LIN {X 0,Y 171.672,Z 289.498,A -85,B 0,C 180,E1 -23440.312,E2 -23440.312} C_VEL
LIN {X 0,Y 173.108,Z 291.829,A -85,B 0,C 180,E1 -23441.183,E2 -23441.183} C_VEL
LIN {X 0,Y 175.242,Z 296.051,A -85,B 0,C 180,E1 -23442.591,E2 -23442.591} C_VEL
LIN {X 0,Y 178.721,Z 304.171,A -85,B 0,C 180,E1 -23445.058,E2 -23445.058} C_VEL
LIN {X 0,Y 180.563,Z 309.956,A -85,B 0,C 180,E1 -23446.66,E2 -23446.66} C_VEL
LIN {X 0,Y 181.625,Z 319.41,A -85,B 0,C 180,E1 -23448.871,E2 -23448.871} C_VEL
LIN {X 0,Y 181.951,Z 330.232,A -85,B 0,C 180,E1 -23451.521,E2 -23451.521} C_VEL
LIN {X 0,Y 181.208,Z 341.103,A -85,B 0,C 180,E1 -23454.43,E2 -23454.43} C_VEL
LIN {X 0,Y 179.983,Z 349.237,A -85,B 0,C 180,E1 -23456.865,E2 -23456.865} C_VEL
LIN {X 0,Y 178.407,Z 354.481,A -85,B 0,C 180,E1 -23458.54,E2 -23458.54} C_VEL
LIN {X 0,Y 174.215,Z 363.38,A -85,B 0,C 180,E1 -23461.709,E2 -23461.709} C_VEL
LIN {X 0,Y 170.995,Z 369.924,A -85,B 0,C 180,E1 -23464.717,E2 -23464.717} C_VEL
LIN {X 0,Y 168.225,Z 375.423,A -85,B 0,C 180,E1 -23467.918,E2 -23467.918} C_VEL
LIN {X 0,Y 165.735,Z 380.164,A -85,B 0,C 180,E1 -23471.46,E2 -23471.46} C_VEL
LIN {X 0,Y 163.854,Z 383.806,A -85,B 0,C 180,E1 -23475.091,E2 -23475.091} C_VEL
LIN {X 0,Y 163.072,Z 385.703,A -85,B 0,C 180,E1 -23477.56,E2 -23477.56} C_VEL
LIN {X 0,Y 162.169,Z 388.175,A -85,B 0,C 180,E1 -23482.533,E2 -23482.533} C_VEL
LIN {X 0,Y 162.078,Z 388.951,A -85,B 0,C 180,E1 -23485.808,E2 -23485.808} C_VEL
LIN {X 0,Y 162.342,Z 388.901,A -85,B 0,C 180,E1 -23490.004,E2 -23490.004} C_VEL
LIN {X 0,Y 162.14,Z 387.508,A -85,B 0,C 180,E1 -23494.483,E2 -23494.483} C_VEL
LIN {X 0,Y 162.204,Z 385.856,A -85,B 0,C 180,E1 -23497.472,E2 -23497.472} C_VEL
LIN {X 0,Y 162.769,Z 382.872,A -85,B 0,C 180,E1 -23501.207,E2 -23501.207} C_VEL
LIN {X 0,Y 163.813,Z 378.83,A -85,B 0,C 180,E1 -23504.92,E2 -23504.92} C_VEL
LIN {X 0,Y 166.011,Z 372.637,A -85,B 0,C 180,E1 -23509.157,E2 -23509.157} C_VEL
LIN {X 0,Y 168.468,Z 365.702,A -85,B 0,C 180,E1 -23512.788,E2 -23512.788} C_VEL
LIN {X 0,Y 170.299,Z 360.479,A -85,B 0,C 180,E1 -23515.028,E2 -23515.028} C_VEL
LIN {X 0,Y 171.171,Z 358.102,A -85,B 0,C 180,E1 -23515.922,E2 -23515.922} C_VEL
LIN {X 0,Y 171.863,Z 354.222,A -85,B 0,C 180,E1 -23517.39,E2 -23517.39} C_VEL
LIN {X 0,Y 171.49,Z 350.309,A -85,B 0,C 180,E1 -23518.883,E2 -23518.883} C_VEL
LIN {X 0,Y 169.685,Z 342.18,A -85,B 0,C 180,E1 -23521.821,E2 -23521.821} C_VEL
LIN {X 0,Y 169.296,Z 337.746,A -85,B 0,C 180,E1 -23523.199,E2 -23523.199} C_VEL
LIN {X 0,Y 169.37,Z 336.183,A -85,B 0,C 180,E1 -23523.629,E2 -23523.629} C_VEL
LIN {X 0,Y 169.918,Z 325.947,A -85,B 0,C 180,E1 -23526.159,E2 -23526.159} C_VEL
LIN {X 0,Y 169.626,Z 314.591,A -85,B 0,C 180,E1 -23528.627,E2 -23528.627} C_VEL
LIN {X 0,Y 168.295,Z 303.304,A -85,B 0,C 180,E1 -23530.881,E2 -23530.881} C_VEL
LIN {X 0,Y 166.877,Z 296.979,A -85,B 0,C 180,E1 -23532.153,E2 -23532.153} C_VEL
LIN {X 0,Y 163.62,Z 289.327,A -85,B 0,C 180,E1 -23534.018,E2 -23534.018} C_VEL
LIN {X 0,Y 161.492,Z 284.949,A -85,B 0,C 180,E1 -23535.128,E2 -23535.128} C_VEL
LIN {X 0,Y 159.84,Z 281.976,A -85,B 0,C 180,E1 -23535.952,E2 -23535.952} C_VEL
LIN {X 0,Y 159.355,Z 280.151,A -85,B 0,C 180,E1 -23536.332,E2 -23536.332} C_VEL
LIN {X 0,Y 158.671,Z 276.748,A -85,B 0,C 180,E1 -23541.677,E2 -23541.677} C_VEL
LIN {X 0,Y 158.331,Z 274.968,A -85,B 0,C 180,E1 -23544.757,E2 -23544.757} C_VEL
LIN {X 0,Y 157.783,Z 271.808,A -85,B 0,C 180,E1 -23550.662,E2 -23550.662} C_VEL
LIN {X 0,Y 157.407,Z 269.136,A -85,B 0,C 180,E1 -23556.307,E2 -23556.307} C_VEL
LIN {X 0,Y 157.365,Z 268.884,A -85,B 0,C 180,E1 -23559.067,E2 -23559.067} C_VEL
LIN {X 0,Y 157.424,Z 268.877,A -85,B 0,C 180,E1 -23564.463,E2 -23564.463} C_VEL
LIN {X 0,Y 157.696,Z 268.844,A -85,B 0,C 180,E1 -23569.731,E2 -23569.731} C_VEL
LIN {X 0,Y 157.773,Z 268.829,A -85,B 0,C 180,E1 -23572.321,E2 -23572.321} C_VEL
LIN {X 0,Y 158.256,Z 268.766,A -85,B 0,C 180,E1 -23580,E2 -23580} C_VEL
LIN {X 0,Y 157.768,Z 268.832,A -85,B 0,C 180,E1 -23587.68,E2 -23587.68} C_VEL
LIN {X 0,Y 157.642,Z 268.846,A -85,B 0,C 180,E1 -23591.227,E2 -23591.227} C_VEL
LIN {X 0,Y 157.428,Z 268.869,A -85,B 0,C 180,E1 -23595.537,E2 -23595.537} C_VEL
LIN {X 0,Y 157.313,Z 268.885,A -85,B 0,C 180,E1 -23600.941,E2 -23600.941} C_VEL
LIN {X 0,Y 157.275,Z 268.895,A -85,B 0,C 180,E1 -23606.648,E2 -23606.648} C_VEL
LIN {X 0,Y 157.276,Z 268.891,A -85,B 0,C 180,E1 -23612.428,E2 -23612.428} C_VEL
LIN {X 0,Y 157.276,Z 268.891,A -85,B 0,C 180,E1 -23616.447,E2 -23616.447} C_VEL
LIN {X 0,Y 157.2,Z 268.903,A -85,B 0,C 180,E1 -23622.115,E2 -23622.115} C_VEL
LIN {X 0,Y 157.242,Z 269.093,A -85,B 0,C 180,E1 -23627.561,E2 -23627.561} C_VEL
LIN {X 0,Y 158.301,Z 271.841,A -85,B 0,C 180,E1 -23628.219,E2 -23628.219} C_VEL
LIN {X 0,Y 160.043,Z 273.99,A -85,B 0,C 180,E1 -23629.056,E2 -23629.056} C_VEL
LIN {X 0,Y 162.024,Z 277.365,A -85,B 0,C 180,E1 -23630.123,E2 -23630.123} C_VEL
LIN {X 0,Y 166.172,Z 285.02,A -85,B 0,C 180,E1 -23632.468,E2 -23632.468} C_VEL
LIN {X 0,Y 169.015,Z 291.893,A -85,B 0,C 180,E1 -23634.394,E2 -23634.394} C_VEL
LIN {X 0,Y 171.62,Z 301.379,A -85,B 0,C 180,E1 -23636.891,E2 -23636.891} C_VEL
LIN {X 0,Y 173.11,Z 310.138,A -85,B 0,C 180,E1 -23639.237,E2 -23639.237} C_VEL
LIN {X 0,Y 173.769,Z 318.596,A -85,B 0,C 180,E1 -23641.622,E2 -23641.622} C_VEL
LIN {X 0,Y 171.201,Z 327.313,A -85,B 0,C 180,E1 -23643.809,E2 -23643.809} C_VEL
LIN {X 0,Y 167.929,Z 336.319,A -85,B 0,C 180,E1 -23646.569,E2 -23646.569} C_VEL
LIN {X 0,Y 164.545,Z 345.089,A -85,B 0,C 180,E1 -23650.016,E2 -23650.016} C_VEL
LIN {X 0,Y 161.778,Z 352.126,A -85,B 0,C 180,E1 -23653.594,E2 -23653.594} C_VEL
LIN {X 0,Y 159.361,Z 357.749,A -85,B 0,C 180,E1 -23657.258,E2 -23657.258} C_VEL
LIN {X 0,Y 157.576,Z 362.176,A -85,B 0,C 180,E1 -23661.016,E2 -23661.016} C_VEL
LIN {X 0,Y 156.24,Z 365.551,A -85,B 0,C 180,E1 -23664.835,E2 -23664.835} C_VEL
LIN {X 0,Y 155.458,Z 368.499,A -85,B 0,C 180,E1 -23669.996,E2 -23669.996} C_VEL
LIN {X 0,Y 155.372,Z 369.393,A -85,B 0,C 180,E1 -23672.589,E2 -23672.589} C_VEL
LIN {X 0,Y 155.479,Z 369.94,A -85,B 0,C 180,E1 -23676.032,E2 -23676.032} C_VEL
LIN {X 0,Y 155.945,Z 369.683,A -85,B 0,C 180,E1 -23680.381,E2 -23680.381} C_VEL
LIN {X 0,Y 156.512,Z 369.016,A -85,B 0,C 180,E1 -23682.971,E2 -23682.971} C_VEL
LIN {X 0,Y 157.336,Z 367.935,A -85,B 0,C 180,E1 -23685.542,E2 -23685.542} C_VEL
LIN {X 0,Y 158.403,Z 366.418,A -85,B 0,C 180,E1 -23688.09,E2 -23688.09} C_VEL
LIN {X 0,Y 160.603,Z 363.348,A -85,B 0,C 180,E1 -23691.833,E2 -23691.833} C_VEL
LIN {X 0,Y 163.269,Z 359.22,A -85,B 0,C 180,E1 -23695.492,E2 -23695.492} C_VEL
LIN {X 0,Y 167.172,Z 352.9,A -85,B 0,C 180,E1 -23699.598,E2 -23699.598} C_VEL
LIN {X 0,Y 171.048,Z 345.979,A -85,B 0,C 180,E1 -23702.98,E2 -23702.98} C_VEL
LIN {X 0,Y 175.423,Z 337.268,A -85,B 0,C 180,E1 -23706.219,E2 -23706.219} C_VEL
LIN {X 0,Y 179.363,Z 328.323,A -85,B 0,C 180,E1 -23708.82,E2 -23708.82} C_VEL
LIN {X 0,Y 179.655,Z 326.596,A -85,B 0,C 180,E1 -23709.372,E2 -23709.372} C_VEL
LIN {X 0,Y 179.152,Z 317.685,A -85,B 0,C 180,E1 -23712.437,E2 -23712.437} C_VEL
LIN {X 0,Y 177.698,Z 308.9,A -85,B 0,C 180,E1 -23715.385,E2 -23715.385} C_VEL
LIN {X 0,Y 175.607,Z 301.826,A -85,B 0,C 180,E1 -23717.854,E2 -23717.854} C_VEL
LIN {X 0,Y 171.735,Z 292.618,A -85,B 0,C 180,E1 -23721.343,E2 -23721.343} C_VEL
LIN {X 0,Y 167.163,Z 284.059,A -85,B 0,C 180,E1 -23724.96,E2 -23724.96} C_VEL
LIN {X 0,Y 164.783,Z 280.149,A -85,B 0,C 180,E1 -23726.784,E2 -23726.784} C_VEL
LIN {X 0,Y 161.938,Z 276.182,A -85,B 0,C 180,E1 -23728.895,E2 -23728.895} C_VEL
LIN {X 0,Y 161.277,Z 274.774,A -85,B 0,C 180,E1 -23729.48,E2 -23729.48} C_VEL
LIN {X 0,Y 158.718,Z 272.463,A -85,B 0,C 180,E1 -23731.304,E2 -23731.304} C_VEL
LIN {X 0,Y 157.479,Z 269.821,A -85,B 0,C 180,E1 -23732.455,E2 -23732.455} C_VEL
LIN {X 0,Y 157.37,Z 269.368,A -85,B 0,C 180,E1 -23732.632,E2 -23732.632} C_VEL
LIN {X 0,Y 157.304,Z 268.891,A -85,B 0,C 180,E1 -23736.29,E2 -23736.29} C_VEL
LIN {X 0,Y 157.402,Z 268.876,A -85,B 0,C 180,E1 -23741.787,E2 -23741.787} C_VEL
LIN {X 0,Y 157.544,Z 268.861,A -85,B 0,C 180,E1 -23747.111,E2 -23747.111} C_VEL
LIN {X 0,Y 157.763,Z 268.835,A -85,B 0,C 180,E1 -23749.735,E2 -23749.735} C_VEL
LIN {X 0,Y 157.815,Z 268.828,A -85,B 0,C 180,E1 -23752.322,E2 -23752.322} C_VEL
LIN {X 0,Y 158.004,Z 268.803,A -85,B 0,C 180,E1 -23757.45,E2 -23757.45} C_VEL
LIN {X 0,Y 158.246,Z 268.772,A -85,B 0,C 180,E1 -23760,E2 -23760} C_VEL
LIN {X 0,Y 157.723,Z 268.862,A -85,B 0,C 180,E1 -23765.113,E2 -23765.113} C_VEL
LIN {X 0,Y 157.962,Z 269.906,A -85,B 0,C 180,E1 -23770.251,E2 -23770.251} C_VEL
LIN {X 0,Y 157.918,Z 271.393,A -85,B 0,C 180,E1 -23775.487,E2 -23775.487} C_VEL
LIN {X 0,Y 158.171,Z 273.297,A -85,B 0,C 180,E1 -23781.09,E2 -23781.09} C_VEL
LIN {X 0,Y 158.588,Z 275.985,A -85,B 0,C 180,E1 -23787.595,E2 -23787.595} C_VEL
LIN {X 0,Y 158.956,Z 278.479,A -85,B 0,C 180,E1 -23792.725,E2 -23792.725} C_VEL
LIN {X 0,Y 160.11,Z 281.618,A -85,B 0,C 180,E1 -23793.767,E2 -23793.767} C_VEL
LIN {X 0,Y 162.377,Z 284.59,A -85,B 0,C 180,E1 -23795.373,E2 -23795.373} C_VEL
LIN {X 0,Y 163.054,Z 285.722,A -85,B 0,C 180,E1 -23795.862,E2 -23795.862} C_VEL
LIN {X 0,Y 164.865,Z 289.444,A -85,B 0,C 180,E1 -23797.29,E2 -23797.29} C_VEL
LIN {X 0,Y 166.299,Z 291.666,A -85,B 0,C 180,E1 -23798.272,E2 -23798.272} C_VEL
LIN {X 0,Y 168.363,Z 295.763,A -85,B 0,C 180,E1 -23799.829,E2 -23799.829} C_VEL
LIN {X 0,Y 171.594,Z 302.812,A -85,B 0,C 180,E1 -23802.316,E2 -23802.316} C_VEL
LIN {X 0,Y 174.732,Z 311.358,A -85,B 0,C 180,E1 -23805.082,E2 -23805.082} C_VEL
LIN {X 0,Y 175.6,Z 316.698,A -85,B 0,C 180,E1 -23806.503,E2 -23806.503} C_VEL
LIN {X 0,Y 176.02,Z 327.827,A -85,B 0,C 180,E1 -23809.342,E2 -23809.342} C_VEL
LIN {X 0,Y 175.468,Z 337.565,A -85,B 0,C 180,E1 -23811.994,E2 -23811.994} C_VEL
LIN {X 0,Y 174.366,Z 346.244,A -85,B 0,C 180,E1 -23814.625,E2 -23814.625} C_VEL
LIN {X 0,Y 172.964,Z 352.639,A -85,B 0,C 180,E1 -23816.737,E2 -23816.737} C_VEL
LIN {X 0,Y 170.1,Z 358.951,A -85,B 0,C 180,E1 -23818.909,E2 -23818.909} C_VEL
LIN {X 0,Y 166.033,Z 366.907,A -85,B 0,C 180,E1 -23822.254,E2 -23822.254} C_VEL
LIN {X 0,Y 162.685,Z 373.292,A -85,B 0,C 180,E1 -23825.774,E2 -23825.774} C_VEL
LIN {X 0,Y 159.795,Z 378.389,A -85,B 0,C 180,E1 -23829.404,E2 -23829.404} C_VEL
LIN {X 0,Y 157.566,Z 382.364,A -85,B 0,C 180,E1 -23833.151,E2 -23833.151} C_VEL
LIN {X 0,Y 156.091,Z 385.326,A -85,B 0,C 180,E1 -23836.994,E2 -23836.994} C_VEL
LIN {X 0,Y 155.109,Z 387.774,A -85,B 0,C 180,E1 -23842.191,E2 -23842.191} C_VEL
LIN {X 0,Y 155.007,Z 388.553,A -85,B 0,C 180,E1 -23845.927,E2 -23845.927} C_VEL
LIN {X 0,Y 155.254,Z 388.457,A -85,B 0,C 180,E1 -23850.004,E2 -23850.004} C_VEL
LIN {X 0,Y 155.075,Z 387.163,A -85,B 0,C 180,E1 -23854.412,E2 -23854.412} C_VEL
LIN {X 0,Y 155.159,Z 385.37,A -85,B 0,C 180,E1 -23857.814,E2 -23857.814} C_VEL
LIN {X 0,Y 155.79,Z 382.365,A -85,B 0,C 180,E1 -23861.716,E2 -23861.716} C_VEL
LIN {X 0,Y 156.919,Z 378.296,A -85,B 0,C 180,E1 -23865.592,E2 -23865.592} C_VEL
LIN {X 0,Y 159.261,Z 372.063,A -85,B 0,C 180,E1 -23870.002,E2 -23870.002} C_VEL
LIN {X 0,Y 161.71,Z 365.444,A -85,B 0,C 180,E1 -23873.606,E2 -23873.606} C_VEL
LIN {X 0,Y 164.999,Z 356.823,A -85,B 0,C 180,E1 -23877.255,E2 -23877.255} C_VEL
LIN {X 0,Y 167.455,Z 349.995,A -85,B 0,C 180,E1 -23879.551,E2 -23879.551} C_VEL
LIN {X 0,Y 168.915,Z 340.714,A -85,B 0,C 180,E1 -23882.394,E2 -23882.394} C_VEL
LIN {X 0,Y 169.37,Z 336.183,A -85,B 0,C 180,E1 -23883.629,E2 -23883.629} C_VEL
LIN {X 0,Y 169.123,Z 331.677,A -85,B 0,C 180,E1 -23884.918,E2 -23884.918} C_VEL
LIN {X 0,Y 166.874,Z 324.632,A -85,B 0,C 180,E1 -23887.172,E2 -23887.172} C_VEL
LIN {X 0,Y 164.677,Z 318.905,A -85,B 0,C 180,E1 -23888.963,E2 -23888.963} C_VEL
LIN {X 0,Y 163.523,Z 314.238,A -85,B 0,C 180,E1 -23890.21,E2 -23890.21} C_VEL
LIN {X 0,Y 163.305,Z 312.574,A -85,B 0,C 180,E1 -23890.589,E2 -23890.589} C_VEL
LIN {X 0,Y 162.2,Z 303.334,A -85,B 0,C 180,E1 -23892.558,E2 -23892.558} C_VEL
LIN {X 0,Y 160.439,Z 297.745,A -85,B 0,C 180,E1 -23893.942,E2 -23893.942} C_VEL
LIN {X 0,Y 156.925,Z 289.667,A -85,B 0,C 180,E1 -23896.148,E2 -23896.148} C_VEL
LIN {X 0,Y 155.023,Z 285.715,A -85,B 0,C 180,E1 -23897.275,E2 -23897.275} C_VEL
LIN {X 0,Y 152.557,Z 281.546,A -85,B 0,C 180,E1 -23898.625,E2 -23898.625} C_VEL
LIN {X 0,Y 151.956,Z 279.532,A -85,B 0,C 180,E1 -23899.094,E2 -23899.094} C_VEL
LIN {X 0,Y 151.576,Z 277.292,A -85,B 0,C 180,E1 -23902.932,E2 -23902.932} C_VEL
LIN {X 0,Y 150.916,Z 273.997,A -85,B 0,C 180,E1 -23909.186,E2 -23909.186} C_VEL
LIN {X 0,Y 150.529,Z 271.205,A -85,B 0,C 180,E1 -23915.153,E2 -23915.153} C_VEL
LIN {X 0,Y 150.327,Z 269.76,A -85,B 0,C 180,E1 -23918.801,E2 -23918.801} C_VEL
LIN {X 0,Y 150.333,Z 269.762,A -85,B 0,C 180,E1 -23923.71,E2 -23923.71} C_VEL
LIN {X 0,Y 150.616,Z 269.726,A -85,B 0,C 180,E1 -23929.243,E2 -23929.243} C_VEL
LIN {X 0,Y 150.711,Z 269.709,A -85,B 0,C 180,E1 -23931.958,E2 -23931.958} C_VEL
LIN {X 0,Y 151.215,Z 269.643,A -85,B 0,C 180,E1 -23940,E2 -23940} C_VEL
LIN {X 0,Y 150.691,Z 269.713,A -85,B 0,C 180,E1 -23948.043,E2 -23948.043} C_VEL
LIN {X 0,Y 150.584,Z 269.726,A -85,B 0,C 180,E1 -23951.43,E2 -23951.43} C_VEL
LIN {X 0,Y 150.333,Z 269.757,A -85,B 0,C 180,E1 -23956.29,E2 -23956.29} C_VEL
LIN {X 0,Y 150.291,Z 269.758,A -85,B 0,C 180,E1 -23960.721,E2 -23960.721} C_VEL
LIN {X 0,Y 150.193,Z 269.776,A -85,B 0,C 180,E1 -23967.236,E2 -23967.236} C_VEL
LIN {X 0,Y 150.217,Z 269.769,A -85,B 0,C 180,E1 -23972.626,E2 -23972.626} C_VEL
LIN {X 0,Y 150.186,Z 269.774,A -85,B 0,C 180,E1 -23977.47,E2 -23977.47} C_VEL
LIN {X 0,Y 150.145,Z 269.783,A -85,B 0,C 180,E1 -23981.497,E2 -23981.497} C_VEL
LIN {X 0,Y 150.132,Z 269.793,A -85,B 0,C 180,E1 -23984.818,E2 -23984.818} C_VEL
LIN {X 0,Y 151.135,Z 272.602,A -85,B 0,C 180,E1 -23985.545,E2 -23985.545} C_VEL
LIN {X 0,Y 153.242,Z 275.172,A -85,B 0,C 180,E1 -23986.696,E2 -23986.696} C_VEL
LIN {X 0,Y 155.261,Z 278.518,A -85,B 0,C 180,E1 -23987.896,E2 -23987.896} C_VEL
LIN {X 0,Y 159.442,Z 285.905,A -85,B 0,C 180,E1 -23990.479,E2 -23990.479} C_VEL
LIN {X 0,Y 163.192,Z 294.405,A -85,B 0,C 180,E1 -23993.16,E2 -23993.16} C_VEL
LIN {X 0,Y 165.754,Z 304.364,A -85,B 0,C 180,E1 -23996,E2 -23996} C_VEL
LIN {X 0,Y 167.084,Z 313.779,A -85,B 0,C 180,E1 -23998.723,E2 -23998.723} C_VEL
LIN {X 0,Y 167.338,Z 320.547,A -85,B 0,C 180,E1 -24000.771,E2 -24000.771} C_VEL
LIN {X 0,Y 164.211,Z 329.985,A -85,B 0,C 180,E1 -24003.292,E2 -24003.292} C_VEL
LIN {X 0,Y 160.844,Z 338.618,A -85,B 0,C 180,E1 -24006.157,E2 -24006.157} C_VEL
LIN {X 0,Y 157.478,Z 346.868,A -85,B 0,C 180,E1 -24009.691,E2 -24009.691} C_VEL
LIN {X 0,Y 154.527,Z 353.718,A -85,B 0,C 180,E1 -24013.482,E2 -24013.482} C_VEL
LIN {X 0,Y 151.754,Z 359.903,A -85,B 0,C 180,E1 -24017.967,E2 -24017.967} C_VEL
LIN {X 0,Y 150.022,Z 363.938,A -85,B 0,C 180,E1 -24021.917,E2 -24021.917} C_VEL
LIN {X 0,Y 149.203,Z 366.048,A -85,B 0,C 180,E1 -24024.59,E2 -24024.59} C_VEL
LIN {X 0,Y 148.393,Z 368.97,A -85,B 0,C 180,E1 -24029.996,E2 -24029.996} C_VEL
LIN {X 0,Y 148.29,Z 369.852,A -85,B 0,C 180,E1 -24032.712,E2 -24032.712} C_VEL
LIN {X 0,Y 148.377,Z 370.348,A -85,B 0,C 180,E1 -24035.907,E2 -24035.907} C_VEL
LIN {X 0,Y 148.947,Z 370.092,A -85,B 0,C 180,E1 -24040.875,E2 -24040.875} C_VEL
LIN {X 0,Y 149.581,Z 369.412,A -85,B 0,C 180,E1 -24043.583,E2 -24043.583} C_VEL
LIN {X 0,Y 150.485,Z 368.305,A -85,B 0,C 180,E1 -24046.269,E2 -24046.269} C_VEL
LIN {X 0,Y 151.634,Z 366.775,A -85,B 0,C 180,E1 -24048.927,E2 -24048.927} C_VEL
LIN {X 0,Y 153.998,Z 363.677,A -85,B 0,C 180,E1 -24052.82,E2 -24052.82} C_VEL
LIN {X 0,Y 156.846,Z 359.518,A -85,B 0,C 180,E1 -24056.616,E2 -24056.616} C_VEL
LIN {X 0,Y 160.997,Z 353.165,A -85,B 0,C 180,E1 -24060.854,E2 -24060.854} C_VEL
LIN {X 0,Y 165.104,Z 346.191,A -85,B 0,C 180,E1 -24064.329,E2 -24064.329} C_VEL
LIN {X 0,Y 169.701,Z 337.433,A -85,B 0,C 180,E1 -24067.647,E2 -24067.647} C_VEL
LIN {X 0,Y 172.997,Z 330.392,A -85,B 0,C 180,E1 -24069.771,E2 -24069.771} C_VEL
LIN {X 0,Y 173.468,Z 328.442,A -85,B 0,C 180,E1 -24070.404,E2 -24070.404} C_VEL
LIN {X 0,Y 173.178,Z 319.713,A -85,B 0,C 180,E1 -24073.617,E2 -24073.617} C_VEL
LIN {X 0,Y 172,Z 311.869,A -85,B 0,C 180,E1 -24076.459,E2 -24076.459} C_VEL
LIN {X 0,Y 170.42,Z 305.944,A -85,B 0,C 180,E1 -24078.713,E2 -24078.713} C_VEL
LIN {X 0,Y 166.952,Z 296.993,A -85,B 0,C 180,E1 -24082.382,E2 -24082.382} C_VEL
LIN {X 0,Y 163.073,Z 289.262,A -85,B 0,C 180,E1 -24085.925,E2 -24085.925} C_VEL
LIN {X 0,Y 160.476,Z 284.822,A -85,B 0,C 180,E1 -24088.203,E2 -24088.203} C_VEL
LIN {X 0,Y 158.469,Z 281.585,A -85,B 0,C 180,E1 -24089.979,E2 -24089.979} C_VEL
LIN {X 0,Y 157.694,Z 280.571,A -85,B 0,C 180,E1 -24090.643,E2 -24090.643} C_VEL
LIN {X 0,Y 155.374,Z 277.702,A -85,B 0,C 180,E1 -24092.636,E2 -24092.636} C_VEL
LIN {X 0,Y 154.407,Z 275.643,A -85,B 0,C 180,E1 -24093.678,E2 -24093.678} C_VEL
LIN {X 0,Y 151.842,Z 273.481,A -85,B 0,C 180,E1 -24095.927,E2 -24095.927} C_VEL
LIN {X 0,Y 150.46,Z 270.803,A -85,B 0,C 180,E1 -24097.515,E2 -24097.515} C_VEL
LIN {X 0,Y 150.336,Z 270.24,A -85,B 0,C 180,E1 -24097.857,E2 -24097.857} C_VEL
LIN {X 0,Y 150.351,Z 269.891,A -85,B 0,C 180,E1 -24100.9,E2 -24100.9} C_VEL
LIN {X 0,Y 150.446,Z 269.743,A -85,B 0,C 180,E1 -24106.492,E2 -24106.492} C_VEL
LIN {X 0,Y 150.679,Z 269.715,A -85,B 0,C 180,E1 -24109.247,E2 -24109.247} C_VEL
LIN {X 0,Y 150.754,Z 269.708,A -85,B 0,C 180,E1 -24111.96,E2 -24111.96} C_VEL
LIN {X 0,Y 150.927,Z 269.685,A -85,B 0,C 180,E1 -24117.331,E2 -24117.331} C_VEL
LIN {X 0,Y 151.209,Z 269.803,A -85,B 0,C 180,E1 -24120,E2 -24120} C_VEL
LIN {X 0,Y 150.991,Z 271.195,A -85,B 0,C 180,E1 -24128.027,E2 -24128.027} C_VEL
LIN {X 0,Y 151.02,Z 272.193,A -85,B 0,C 180,E1 -24132.259,E2 -24132.259} C_VEL
LIN {X 0,Y 151.147,Z 274.23,A -85,B 0,C 180,E1 -24138.995,E2 -24138.995} C_VEL
LIN {X 0,Y 151.43,Z 276.319,A -85,B 0,C 180,E1 -24144.689,E2 -24144.689} C_VEL
LIN {X 0,Y 151.662,Z 277.586,A -85,B 0,C 180,E1 -24147.693,E2 -24147.693} C_VEL
LIN {X 0,Y 152.652,Z 280.447,A -85,B 0,C 180,E1 -24148.845,E2 -24148.845} C_VEL
LIN {X 0,Y 154.921,Z 283.56,A -85,B 0,C 180,E1 -24150.877,E2 -24150.877} C_VEL
LIN {X 0,Y 155.929,Z 284.728,A -85,B 0,C 180,E1 -24151.693,E2 -24151.693} C_VEL
LIN {X 0,Y 157.57,Z 288.461,A -85,B 0,C 180,E1 -24153.303,E2 -24153.303} C_VEL
LIN {X 0,Y 159.432,Z 291.108,A -85,B 0,C 180,E1 -24154.777,E2 -24154.777} C_VEL
LIN {X 0,Y 161.439,Z 295.308,A -85,B 0,C 180,E1 -24156.574,E2 -24156.574} C_VEL
LIN {X 0,Y 162.344,Z 296.942,A -85,B 0,C 180,E1 -24157.306,E2 -24157.306} C_VEL
LIN {X 0,Y 165.552,Z 304.184,A -85,B 0,C 180,E1 -24160.176,E2 -24160.176} C_VEL
LIN {X 0,Y 168.337,Z 311.392,A -85,B 0,C 180,E1 -24162.834,E2 -24162.834} C_VEL
LIN {X 0,Y 169.856,Z 317.061,A -85,B 0,C 180,E1 -24164.7,E2 -24164.7} C_VEL
LIN {X 0,Y 170.178,Z 325.932,A -85,B 0,C 180,E1 -24167.102,E2 -24167.102} C_VEL
LIN {X 0,Y 169.814,Z 335.14,A -85,B 0,C 180,E1 -24169.726,E2 -24169.726} C_VEL
LIN {X 0,Y 168.441,Z 345.291,A -85,B 0,C 180,E1 -24172.879,E2 -24172.879} C_VEL
LIN {X 0,Y 166.88,Z 352.441,A -85,B 0,C 180,E1 -24175.356,E2 -24175.356} C_VEL
LIN {X 0,Y 164.86,Z 357.242,A -85,B 0,C 180,E1 -24177.08,E2 -24177.08} C_VEL
LIN {X 0,Y 160.41,Z 365.418,A -85,B 0,C 180,E1 -24180.474,E2 -24180.474} C_VEL
LIN {X 0,Y 157.261,Z 371.005,A -85,B 0,C 180,E1 -24183.459,E2 -24183.459} C_VEL
LIN {X 0,Y 154.054,Z 376.489,A -85,B 0,C 180,E1 -24187.188,E2 -24187.188} C_VEL
LIN {X 0,Y 151.489,Z 380.801,A -85,B 0,C 180,E1 -24191.054,E2 -24191.054} C_VEL
LIN {X 0,Y 150.09,Z 383.097,A -85,B 0,C 180,E1 -24193.687,E2 -24193.687} C_VEL
LIN {X 0,Y 149.133,Z 384.948,A -85,B 0,C 180,E1 -24196.375,E2 -24196.375} C_VEL
LIN {X 0,Y 148.042,Z 387.373,A -85,B 0,C 180,E1 -24201.816,E2 -24201.816} C_VEL
LIN {X 0,Y 147.939,Z 388.156,A -85,B 0,C 180,E1 -24206.054,E2 -24206.054} C_VEL
LIN {X 0,Y 148.168,Z 388.013,A -85,B 0,C 180,E1 -24210.004,E2 -24210.004} C_VEL
LIN {X 0,Y 147.991,Z 386.862,A -85,B 0,C 180,E1 -24214.228,E2 -24214.228} C_VEL
LIN {X 0,Y 148.093,Z 384.879,A -85,B 0,C 180,E1 -24218.189,E2 -24218.189} C_VEL
LIN {X 0,Y 148.786,Z 381.851,A -85,B 0,C 180,E1 -24222.276,E2 -24222.276} C_VEL
LIN {X 0,Y 150.054,Z 377.758,A -85,B 0,C 180,E1 -24226.325,E2 -24226.325} C_VEL
LIN {X 0,Y 152.528,Z 371.485,A -85,B 0,C 180,E1 -24230.926,E2 -24230.926} C_VEL
LIN {X 0,Y 154.789,Z 365.901,A -85,B 0,C 180,E1 -24234.123,E2 -24234.123} C_VEL
LIN {X 0,Y 156.356,Z 361.818,A -85,B 0,C 180,E1 -24236.096,E2 -24236.096} C_VEL
LIN {X 0,Y 159.954,Z 352.877,A -85,B 0,C 180,E1 -24239.628,E2 -24239.628} C_VEL
LIN {X 0,Y 161.145,Z 349.295,A -85,B 0,C 180,E1 -24240.831,E2 -24240.831} C_VEL
LIN {X 0,Y 162.618,Z 339.938,A -85,B 0,C 180,E1 -24243.813,E2 -24243.813} C_VEL
LIN {X 0,Y 163.553,Z 329.5,A -85,B 0,C 180,E1 -24246.651,E2 -24246.651} C_VEL
LIN {X 0,Y 163.643,Z 318.065,A -85,B 0,C 180,E1 -24249.372,E2 -24249.372} C_VEL
LIN {X 0,Y 163.305,Z 312.574,A -85,B 0,C 180,E1 -24250.589,E2 -24250.589} C_VEL
LIN {X 0,Y 162.672,Z 309.405,A -85,B 0,C 180,E1 -24251.375,E2 -24251.375} C_VEL
LIN {X 0,Y 160.725,Z 305.247,A -85,B 0,C 180,E1 -24252.704,E2 -24252.704} C_VEL
LIN {X 0,Y 158.118,Z 301.619,A -85,B 0,C 180,E1 -24254.135,E2 -24254.135} C_VEL
LIN {X 0,Y 152.492,Z 294.366,A -85,B 0,C 180,E1 -24257.13,E2 -24257.13} C_VEL
LIN {X 0,Y 150.966,Z 291.539,A -85,B 0,C 180,E1 -24258.072,E2 -24258.072} C_VEL
LIN {X 0,Y 149.674,Z 289.051,A -85,B 0,C 180,E1 -24258.9,E2 -24258.9} C_VEL
LIN {X 0,Y 147.872,Z 285.19,A -85,B 0,C 180,E1 -24260.127,E2 -24260.127} C_VEL
LIN {X 0,Y 145.314,Z 281.196,A -85,B 0,C 180,E1 -24261.694,E2 -24261.694} C_VEL
LIN {X 0,Y 144.668,Z 278.923,A -85,B 0,C 180,E1 -24262.28,E2 -24262.28} C_VEL
LIN {X 0,Y 144.086,Z 276.201,A -85,B 0,C 180,E1 -24267.552,E2 -24267.552} C_VEL
LIN {X 0,Y 143.648,Z 273.294,A -85,B 0,C 180,E1 -24273.876,E2 -24273.876} C_VEL
LIN {X 0,Y 143.33,Z 270.88,A -85,B 0,C 180,E1 -24279.926,E2 -24279.926} C_VEL
LIN {X 0,Y 143.273,Z 270.639,A -85,B 0,C 180,E1 -24282.884,E2 -24282.884} C_VEL
LIN {X 0,Y 143.542,Z 270.608,A -85,B 0,C 180,E1 -24288.706,E2 -24288.706} C_VEL
LIN {X 0,Y 143.632,Z 270.592,A -85,B 0,C 180,E1 -24291.559,E2 -24291.559} C_VEL
LIN {X 0,Y 144.172,Z 270.52,A -85,B 0,C 180,E1 -24300,E2 -24300} C_VEL
LIN {X 0,Y 143.616,Z 270.592,A -85,B 0,C 180,E1 -24308.442,E2 -24308.442} C_VEL
LIN {X 0,Y 143.51,Z 270.608,A -85,B 0,C 180,E1 -24311.618,E2 -24311.618} C_VEL
LIN {X 0,Y 143.27,Z 270.64,A -85,B 0,C 180,E1 -24317.118,E2 -24317.118} C_VEL
LIN {X 0,Y 143.228,Z 270.641,A -85,B 0,C 180,E1 -24321.193,E2 -24321.193} C_VEL
LIN {X 0,Y 143.151,Z 270.651,A -85,B 0,C 180,E1 -24327.898,E2 -24327.898} C_VEL
LIN {X 0,Y 143.148,Z 270.649,A -85,B 0,C 180,E1 -24333.415,E2 -24333.415} C_VEL
LIN {X 0,Y 143.065,Z 270.661,A -85,B 0,C 180,E1 -24339.69,E2 -24339.69} C_VEL
LIN {X 0,Y 143.114,Z 270.73,A -85,B 0,C 180,E1 -24341.697,E2 -24341.697} C_VEL
LIN {X 0,Y 143.928,Z 273.29,A -85,B 0,C 180,E1 -24342.409,E2 -24342.409} C_VEL
LIN {X 0,Y 145.881,Z 275.494,A -85,B 0,C 180,E1 -24343.616,E2 -24343.616} C_VEL
LIN {X 0,Y 148.362,Z 279.492,A -85,B 0,C 180,E1 -24345.281,E2 -24345.281} C_VEL
LIN {X 0,Y 149.478,Z 281.345,A -85,B 0,C 180,E1 -24346.048,E2 -24346.048} C_VEL
LIN {X 0,Y 152.84,Z 287.147,A -85,B 0,C 180,E1 -24348.351,E2 -24348.351} C_VEL
LIN {X 0,Y 156.345,Z 294.484,A -85,B 0,C 180,E1 -24350.995,E2 -24350.995} C_VEL
LIN {X 0,Y 158.088,Z 299.409,A -85,B 0,C 180,E1 -24352.623,E2 -24352.623} C_VEL
LIN {X 0,Y 160.107,Z 308.638,A -85,B 0,C 180,E1 -24355.486,E2 -24355.486} C_VEL
LIN {X 0,Y 160.998,Z 317.978,A -85,B 0,C 180,E1 -24358.406,E2 -24358.406} C_VEL
LIN {X 0,Y 161.099,Z 321.365,A -85,B 0,C 180,E1 -24359.522,E2 -24359.522} C_VEL
LIN {X 0,Y 158.654,Z 328.792,A -85,B 0,C 180,E1 -24361.559,E2 -24361.559} C_VEL
LIN {X 0,Y 155.08,Z 337.693,A -85,B 0,C 180,E1 -24364.495,E2 -24364.495} C_VEL
LIN {X 0,Y 151.207,Z 346.744,A -85,B 0,C 180,E1 -24368.372,E2 -24368.372} C_VEL
LIN {X 0,Y 147.781,Z 354.305,A -85,B 0,C 180,E1 -24372.705,E2 -24372.705} C_VEL
LIN {X 0,Y 144.854,Z 360.458,A -85,B 0,C 180,E1 -24377.385,E2 -24377.385} C_VEL
LIN {X 0,Y 143.031,Z 364.463,A -85,B 0,C 180,E1 -24381.519,E2 -24381.519} C_VEL
LIN {X 0,Y 142.17,Z 366.546,A -85,B 0,C 180,E1 -24384.322,E2 -24384.322} C_VEL
LIN {X 0,Y 141.328,Z 369.441,A -85,B 0,C 180,E1 -24389.996,E2 -24389.996} C_VEL
LIN {X 0,Y 141.211,Z 370.308,A -85,B 0,C 180,E1 -24392.849,E2 -24392.849} C_VEL
LIN {X 0,Y 141.297,Z 370.76,A -85,B 0,C 180,E1 -24395.85,E2 -24395.85} C_VEL
LIN {X 0,Y 141.955,Z 370.502,A -85,B 0,C 180,E1 -24401.418,E2 -24401.418} C_VEL
LIN {X 0,Y 142.663,Z 369.807,A -85,B 0,C 180,E1 -24404.255,E2 -24404.255} C_VEL
LIN {X 0,Y 143.645,Z 368.675,A -85,B 0,C 180,E1 -24407.067,E2 -24407.067} C_VEL
LIN {X 0,Y 144.899,Z 367.132,A -85,B 0,C 180,E1 -24409.843,E2 -24409.843} C_VEL
LIN {X 0,Y 147.445,Z 364.006,A -85,B 0,C 180,E1 -24413.896,E2 -24413.896} C_VEL
LIN {X 0,Y 150.493,Z 359.817,A -85,B 0,C 180,E1 -24417.835,E2 -24417.835} C_VEL
LIN {X 0,Y 154.915,Z 353.432,A -85,B 0,C 180,E1 -24422.208,E2 -24422.208} C_VEL
LIN {X 0,Y 159.274,Z 346.401,A -85,B 0,C 180,E1 -24425.774,E2 -24425.774} C_VEL
LIN {X 0,Y 164.09,Z 337.6,A -85,B 0,C 180,E1 -24429.174,E2 -24429.174} C_VEL
LIN {X 0,Y 166.671,Z 332.4,A -85,B 0,C 180,E1 -24430.813,E2 -24430.813} C_VEL
LIN {X 0,Y 167.32,Z 330.496,A -85,B 0,C 180,E1 -24431.416,E2 -24431.416} C_VEL
LIN {X 0,Y 167.321,Z 322.867,A -85,B 0,C 180,E1 -24434.434,E2 -24434.434} C_VEL
LIN {X 0,Y 166.4,Z 315.113,A -85,B 0,C 180,E1 -24437.485,E2 -24437.485} C_VEL
LIN {X 0,Y 164.725,Z 308.535,A -85,B 0,C 180,E1 -24440.209,E2 -24440.209} C_VEL
LIN {X 0,Y 161.839,Z 300.594,A -85,B 0,C 180,E1 -24443.783,E2 -24443.783} C_VEL
LIN {X 0,Y 159.146,Z 294.821,A -85,B 0,C 180,E1 -24446.646,E2 -24446.646} C_VEL
LIN {X 0,Y 156.857,Z 290.574,A -85,B 0,C 180,E1 -24448.985,E2 -24448.985} C_VEL
LIN {X 0,Y 154.258,Z 286.367,A -85,B 0,C 180,E1 -24451.605,E2 -24451.605} C_VEL
LIN {X 0,Y 152.128,Z 283.217,A -85,B 0,C 180,E1 -24453.783,E2 -24453.783} C_VEL
LIN {X 0,Y 151.474,Z 281.878,A -85,B 0,C 180,E1 -24454.584,E2 -24454.584} C_VEL
LIN {X 0,Y 149.227,Z 279.589,A -85,B 0,C 180,E1 -24456.861,E2 -24456.861} C_VEL
LIN {X 0,Y 147.772,Z 276.734,A -85,B 0,C 180,E1 -24458.8,E2 -24458.8} C_VEL
LIN {X 0,Y 144.693,Z 274.141,A -85,B 0,C 180,E1 -24462.51,E2 -24462.51} C_VEL
LIN {X 0,Y 143.505,Z 271.609,A -85,B 0,C 180,E1 -24464.556,E2 -24464.556} C_VEL
LIN {X 0,Y 143.457,Z 271.335,A -85,B 0,C 180,E1 -24465.096,E2 -24465.096} C_VEL
LIN {X 0,Y 143.7,Z 271.158,A -85,B 0,C 180,E1 -24468.718,E2 -24468.718} C_VEL
LIN {X 0,Y 143.769,Z 271.156,A -85,B 0,C 180,E1 -24471.567,E2 -24471.567} C_VEL
LIN {X 0,Y 144.025,Z 271.397,A -85,B 0,C 180,E1 -24477.203,E2 -24477.203} C_VEL
LIN {X 0,Y 144.331,Z 271.606,A -85,B 0,C 180,E1 -24480,E2 -24480} C_VEL
LIN {X 0,Y 144.098,Z 273.036,A -85,B 0,C 180,E1 -24488.413,E2 -24488.413} C_VEL
LIN {X 0,Y 144.113,Z 274.074,A -85,B 0,C 180,E1 -24492.77,E2 -24492.77} C_VEL
LIN {X 0,Y 144.13,Z 275.273,A -85,B 0,C 180,E1 -24497.012,E2 -24497.012} C_VEL
LIN {X 0,Y 144.323,Z 276.57,A -85,B 0,C 180,E1 -24500.72,E2 -24500.72} C_VEL
LIN {X 0,Y 145.754,Z 280.144,A -85,B 0,C 180,E1 -24502.971,E2 -24502.971} C_VEL
LIN {X 0,Y 148.748,Z 283.606,A -85,B 0,C 180,E1 -24506.348,E2 -24506.348} C_VEL
LIN {X 0,Y 150.902,Z 288.221,A -85,B 0,C 180,E1 -24508.945,E2 -24508.945} C_VEL
LIN {X 0,Y 152.739,Z 290.649,A -85,B 0,C 180,E1 -24510.694,E2 -24510.694} C_VEL
LIN {X 0,Y 154.454,Z 294.581,A -85,B 0,C 180,E1 -24512.61,E2 -24512.61} C_VEL
LIN {X 0,Y 155.587,Z 296.14,A -85,B 0,C 180,E1 -24513.596,E2 -24513.596} C_VEL
LIN {X 0,Y 157.339,Z 300.365,A -85,B 0,C 180,E1 -24515.498,E2 -24515.498} C_VEL
LIN {X 0,Y 158.581,Z 303.107,A -85,B 0,C 180,E1 -24516.749,E2 -24516.749} C_VEL
LIN {X 0,Y 161.605,Z 310.426,A -85,B 0,C 180,E1 -24519.901,E2 -24519.901} C_VEL
LIN {X 0,Y 163.761,Z 317.26,A -85,B 0,C 180,E1 -24522.526,E2 -24522.526} C_VEL
LIN {X 0,Y 164.49,Z 321.24,A -85,B 0,C 180,E1 -24523.885,E2 -24523.885} C_VEL
LIN {X 0,Y 164.227,Z 332.533,A -85,B 0,C 180,E1 -24527.215,E2 -24527.215} C_VEL
LIN {X 0,Y 163.082,Z 341.721,A -85,B 0,C 180,E1 -24530.109,E2 -24530.109} C_VEL
LIN {X 0,Y 161.343,Z 350.494,A -85,B 0,C 180,E1 -24533.211,E2 -24533.211} C_VEL
LIN {X 0,Y 159.686,Z 355.519,A -85,B 0,C 180,E1 -24535.105,E2 -24535.105} C_VEL
LIN {X 0,Y 154.956,Z 363.923,A -85,B 0,C 180,E1 -24538.566,E2 -24538.566} C_VEL
LIN {X 0,Y 150.91,Z 370.719,A -85,B 0,C 180,E1 -24542.249,E2 -24542.249} C_VEL
LIN {X 0,Y 147.514,Z 376.175,A -85,B 0,C 180,E1 -24546.116,E2 -24546.116} C_VEL
LIN {X 0,Y 144.749,Z 380.459,A -85,B 0,C 180,E1 -24550.135,E2 -24550.135} C_VEL
LIN {X 0,Y 143.25,Z 382.743,A -85,B 0,C 180,E1 -24552.885,E2 -24552.885} C_VEL
LIN {X 0,Y 142.204,Z 384.57,A -85,B 0,C 180,E1 -24555.698,E2 -24555.698} C_VEL
LIN {X 0,Y 141.003,Z 386.972,A -85,B 0,C 180,E1 -24561.405,E2 -24561.405} C_VEL
LIN {X 0,Y 140.868,Z 387.759,A -85,B 0,C 180,E1 -24566.21,E2 -24566.21} C_VEL
LIN {X 0,Y 141.082,Z 387.569,A -85,B 0,C 180,E1 -24570.004,E2 -24570.004} C_VEL
LIN {X 0,Y 140.898,Z 386.581,A -85,B 0,C 180,E1 -24573.971,E2 -24573.971} C_VEL
LIN {X 0,Y 141.046,Z 384.386,A -85,B 0,C 180,E1 -24578.601,E2 -24578.601} C_VEL
LIN {X 0,Y 141.802,Z 381.334,A -85,B 0,C 180,E1 -24582.891,E2 -24582.891} C_VEL
LIN {X 0,Y 143.214,Z 377.216,A -85,B 0,C 180,E1 -24587.128,E2 -24587.128} C_VEL
LIN {X 0,Y 145.841,Z 370.907,A -85,B 0,C 180,E1 -24591.934,E2 -24591.934} C_VEL
LIN {X 0,Y 148.193,Z 365.285,A -85,B 0,C 180,E1 -24595.27,E2 -24595.27} C_VEL
LIN {X 0,Y 151.779,Z 357.047,A -85,B 0,C 180,E1 -24599.095,E2 -24599.095} C_VEL
LIN {X 0,Y 154.39,Z 350.418,A -85,B 0,C 180,E1 -24601.571,E2 -24601.571} C_VEL
LIN {X 0,Y 156.086,Z 341.382,A -85,B 0,C 180,E1 -24604.647,E2 -24604.647} C_VEL
LIN {X 0,Y 157.22,Z 331.565,A -85,B 0,C 180,E1 -24607.525,E2 -24607.525} C_VEL
LIN {X 0,Y 157.615,Z 321.263,A -85,B 0,C 180,E1 -24610.193,E2 -24610.193} C_VEL
LIN {X 0,Y 157.063,Z 310.399,A -85,B 0,C 180,E1 -24612.777,E2 -24612.777} C_VEL
LIN {X 0,Y 156.089,Z 303.967,A -85,B 0,C 180,E1 -24614.307,E2 -24614.307} C_VEL
LIN {X 0,Y 152.367,Z 294.394,A -85,B 0,C 180,E1 -24617.13,E2 -24617.13} C_VEL
LIN {X 0,Y 150.966,Z 291.539,A -85,B 0,C 180,E1 -24618.072,E2 -24618.072} C_VEL
LIN {X 0,Y 149.274,Z 289.105,A -85,B 0,C 180,E1 -24619.053,E2 -24619.053} C_VEL
LIN {X 0,Y 147.106,Z 287.44,A -85,B 0,C 180,E1 -24620.169,E2 -24620.169} C_VEL
LIN {X 0,Y 140.124,Z 283.641,A -85,B 0,C 180,E1 -24623.886,E2 -24623.886} C_VEL
LIN {X 0,Y 139.461,Z 283.022,A -85,B 0,C 180,E1 -24624.304,E2 -24624.304} C_VEL
LIN {X 0,Y 137.728,Z 279.917,A -85,B 0,C 180,E1 -24625.631,E2 -24625.631} C_VEL
LIN {X 0,Y 137.252,Z 278.236,A -85,B 0,C 180,E1 -24626.162,E2 -24626.162} C_VEL
LIN {X 0,Y 136.78,Z 275.401,A -85,B 0,C 180,E1 -24632.456,E2 -24632.456} C_VEL
LIN {X 0,Y 136.466,Z 272.846,A -85,B 0,C 180,E1 -24638.869,E2 -24638.869} C_VEL
LIN {X 0,Y 136.271,Z 271.802,A -85,B 0,C 180,E1 -24641.975,E2 -24641.975} C_VEL
LIN {X 0,Y 136.435,Z 271.493,A -85,B 0,C 180,E1 -24648.179,E2 -24648.179} C_VEL
LIN {X 0,Y 136.557,Z 271.476,A -85,B 0,C 180,E1 -24651.119,E2 -24651.119} C_VEL
LIN {X 0,Y 137.128,Z 271.397,A -85,B 0,C 180,E1 -24660,E2 -24660} C_VEL
LIN {X 0,Y 136.546,Z 271.47,A -85,B 0,C 180,E1 -24668.883,E2 -24668.883} C_VEL
LIN {X 0,Y 136.424,Z 271.492,A -85,B 0,C 180,E1 -24671.892,E2 -24671.892} C_VEL
LIN {X 0,Y 136.18,Z 271.521,A -85,B 0,C 180,E1 -24678.039,E2 -24678.039} C_VEL
LIN {X 0,Y 136.152,Z 271.525,A -85,B 0,C 180,E1 -24681.689,E2 -24681.689} C_VEL
LIN {X 0,Y 136.071,Z 271.53,A -85,B 0,C 180,E1 -24688.584,E2 -24688.584} C_VEL
LIN {X 0,Y 136.05,Z 271.537,A -85,B 0,C 180,E1 -24694.628,E2 -24694.628} C_VEL
LIN {X 0,Y 136.054,Z 271.589,A -85,B 0,C 180,E1 -24697.955,E2 -24697.955} C_VEL
LIN {X 0,Y 136.928,Z 274.224,A -85,B 0,C 180,E1 -24698.836,E2 -24698.836} C_VEL
LIN {X 0,Y 138.976,Z 276.433,A -85,B 0,C 180,E1 -24700.317,E2 -24700.317} C_VEL
LIN {X 0,Y 139.584,Z 277.325,A -85,B 0,C 180,E1 -24700.788,E2 -24700.788} C_VEL
LIN {X 0,Y 141.333,Z 280.339,A -85,B 0,C 180,E1 -24702.167,E2 -24702.167} C_VEL
LIN {X 0,Y 142.63,Z 282.151,A -85,B 0,C 180,E1 -24703.132,E2 -24703.132} C_VEL
LIN {X 0,Y 146.417,Z 288.596,A -85,B 0,C 180,E1 -24706.055,E2 -24706.055} C_VEL
LIN {X 0,Y 150.345,Z 296.596,A -85,B 0,C 180,E1 -24709.328,E2 -24709.328} C_VEL
LIN {X 0,Y 152.49,Z 302.76,A -85,B 0,C 180,E1 -24711.583,E2 -24711.583} C_VEL
LIN {X 0,Y 154.215,Z 311.681,A -85,B 0,C 180,E1 -24714.582,E2 -24714.582} C_VEL
LIN {X 0,Y 154.788,Z 319.986,A -85,B 0,C 180,E1 -24717.368,E2 -24717.368} C_VEL
LIN {X 0,Y 154.826,Z 323.303,A -85,B 0,C 180,E1 -24718.528,E2 -24718.528} C_VEL
LIN {X 0,Y 150.968,Z 333.286,A -85,B 0,C 180,E1 -24721.495,E2 -24721.495} C_VEL
LIN {X 0,Y 147.384,Z 341.46,A -85,B 0,C 180,E1 -24724.581,E2 -24724.581} C_VEL
LIN {X 0,Y 144.048,Z 348.72,A -85,B 0,C 180,E1 -24728.078,E2 -24728.078} C_VEL
LIN {X 0,Y 141.065,Z 354.89,A -85,B 0,C 180,E1 -24731.853,E2 -24731.853} C_VEL
LIN {X 0,Y 137.973,Z 361.009,A -85,B 0,C 180,E1 -24736.745,E2 -24736.745} C_VEL
LIN {X 0,Y 136.048,Z 364.986,A -85,B 0,C 180,E1 -24741.08,E2 -24741.08} C_VEL
LIN {X 0,Y 135.142,Z 367.042,A -85,B 0,C 180,E1 -24744.026,E2 -24744.026} C_VEL
LIN {X 0,Y 134.264,Z 369.911,A -85,B 0,C 180,E1 -24749.996,E2 -24749.996} C_VEL
LIN {X 0,Y 134.136,Z 370.76,A -85,B 0,C 180,E1 -24752.999,E2 -24752.999} C_VEL
LIN {X 0,Y 134.23,Z 371.185,A -85,B 0,C 180,E1 -24756.006,E2 -24756.006} C_VEL
LIN {X 0,Y 134.506,Z 371.235,A -85,B 0,C 180,E1 -24759.014,E2 -24759.014} C_VEL
LIN {X 0,Y 135.759,Z 370.199,A -85,B 0,C 180,E1 -24764.997,E2 -24764.997} C_VEL
LIN {X 0,Y 136.843,Z 369.046,A -85,B 0,C 180,E1 -24767.943,E2 -24767.943} C_VEL
LIN {X 0,Y 138.211,Z 367.49,A -85,B 0,C 180,E1 -24770.847,E2 -24770.847} C_VEL
LIN {X 0,Y 140.933,Z 364.336,A -85,B 0,C 180,E1 -24775.075,E2 -24775.075} C_VEL
LIN {X 0,Y 144.209,Z 360.118,A -85,B 0,C 180,E1 -24779.162,E2 -24779.162} C_VEL
LIN {X 0,Y 148.913,Z 353.696,A -85,B 0,C 180,E1 -24783.674,E2 -24783.674} C_VEL
LIN {X 0,Y 153.531,Z 346.612,A -85,B 0,C 180,E1 -24787.334,E2 -24787.334} C_VEL
LIN {X 0,Y 158.619,Z 337.767,A -85,B 0,C 180,E1 -24790.803,E2 -24790.803} C_VEL
LIN {X 0,Y 161.214,Z 332.554,A -85,B 0,C 180,E1 -24792.502,E2 -24792.502} C_VEL
LIN {X 0,Y 161.392,Z 324.705,A -85,B 0,C 180,E1 -24795.833,E2 -24795.833} C_VEL
LIN {X 0,Y 160.622,Z 317.295,A -85,B 0,C 180,E1 -24798.979,E2 -24798.979} C_VEL
LIN {X 0,Y 158.699,Z 309.857,A -85,B 0,C 180,E1 -24802.43,E2 -24802.43} C_VEL
LIN {X 0,Y 156.263,Z 303.197,A -85,B 0,C 180,E1 -24805.792,E2 -24805.792} C_VEL
LIN {X 0,Y 153.145,Z 296.295,A -85,B 0,C 180,E1 -24809.681,E2 -24809.681} C_VEL
LIN {X 0,Y 150.945,Z 292.448,A -85,B 0,C 180,E1 -24812.25,E2 -24812.25} C_VEL
LIN {X 0,Y 148.809,Z 288.818,A -85,B 0,C 180,E1 -24814.845,E2 -24814.845} C_VEL
LIN {X 0,Y 145.76,Z 284.462,A -85,B 0,C 180,E1 -24818.707,E2 -24818.707} C_VEL
LIN {X 0,Y 145.335,Z 283.274,A -85,B 0,C 180,E1 -24819.476,E2 -24819.476} C_VEL
LIN {X 0,Y 142.534,Z 280.551,A -85,B 0,C 180,E1 -24823.345,E2 -24823.345} C_VEL
LIN {X 0,Y 141.432,Z 278.115,A -85,B 0,C 180,E1 -24825.613,E2 -24825.613} C_VEL
LIN {X 0,Y 137.379,Z 274.212,A -85,B 0,C 180,E1 -24836.15,E2 -24836.15} C_VEL
LIN {X 0,Y 137.243,Z 273.254,A -85,B 0,C 180,E1 -24838.166,E2 -24838.166} C_VEL
LIN {X 0,Y 137.456,Z 273.387,A -85,B 0,C 180,E1 -24840,E2 -24840} C_VEL
LIN {X 0,Y 137.195,Z 274.666,A -85,B 0,C 180,E1 -24846.618,E2 -24846.618} C_VEL
LIN {X 0,Y 139.099,Z 279.546,A -85,B 0,C 180,E1 -24854.109,E2 -24854.109} C_VEL
LIN {X 0,Y 142.254,Z 283.276,A -85,B 0,C 180,E1 -24859.856,E2 -24859.856} C_VEL
LIN {X 0,Y 143.796,Z 287.104,A -85,B 0,C 180,E1 -24862.636,E2 -24862.636} C_VEL
LIN {X 0,Y 146.202,Z 290.287,A -85,B 0,C 180,E1 -24865.709,E2 -24865.709} C_VEL
LIN {X 0,Y 147.954,Z 294.353,A -85,B 0,C 180,E1 -24868.167,E2 -24868.167} C_VEL
LIN {X 0,Y 149.289,Z 296.24,A -85,B 0,C 180,E1 -24869.624,E2 -24869.624} C_VEL
LIN {X 0,Y 150.786,Z 300.073,A -85,B 0,C 180,E1 -24871.625,E2 -24871.625} C_VEL
LIN {X 0,Y 151.963,Z 302.229,A -85,B 0,C 180,E1 -24872.916,E2 -24872.916} C_VEL
LIN {X 0,Y 155.605,Z 311.487,A -85,B 0,C 180,E1 -24877.412,E2 -24877.412} C_VEL
LIN {X 0,Y 158.135,Z 319.648,A -85,B 0,C 180,E1 -24880.934,E2 -24880.934} C_VEL
LIN {X 0,Y 158.979,Z 324.011,A -85,B 0,C 180,E1 -24882.612,E2 -24882.612} C_VEL
LIN {X 0,Y 158.478,Z 333.757,A -85,B 0,C 180,E1 -24885.713,E2 -24885.713} C_VEL
LIN {X 0,Y 157.202,Z 342.505,A -85,B 0,C 180,E1 -24888.656,E2 -24888.656} C_VEL
LIN {X 0,Y 154.937,Z 352.037,A -85,B 0,C 180,E1 -24892.244,E2 -24892.244} C_VEL
LIN {X 0,Y 153.048,Z 356.81,A -85,B 0,C 180,E1 -24894.168,E2 -24894.168} C_VEL
LIN {X 0,Y 148.161,Z 364.912,A -85,B 0,C 180,E1 -24897.753,E2 -24897.753} C_VEL
LIN {X 0,Y 143.693,Z 371.885,A -85,B 0,C 180,E1 -24901.883,E2 -24901.883} C_VEL
LIN {X 0,Y 139.922,Z 377.402,A -85,B 0,C 180,E1 -24906.313,E2 -24906.313} C_VEL
LIN {X 0,Y 137.216,Z 381.302,A -85,B 0,C 180,E1 -24910.559,E2 -24910.559} C_VEL
LIN {X 0,Y 135.306,Z 384.192,A -85,B 0,C 180,E1 -24914.952,E2 -24914.952} C_VEL
LIN {X 0,Y 133.963,Z 386.572,A -85,B 0,C 180,E1 -24920.949,E2 -24920.949} C_VEL
LIN {X 0,Y 133.786,Z 387.365,A -85,B 0,C 180,E1 -24926.468,E2 -24926.468} C_VEL
LIN {X 0,Y 133.999,Z 387.126,A -85,B 0,C 180,E1 -24930.004,E2 -24930.004} C_VEL
LIN {X 0,Y 133.81,Z 386.281,A -85,B 0,C 180,E1 -24933.694,E2 -24933.694} C_VEL
LIN {X 0,Y 133.999,Z 383.892,A -85,B 0,C 180,E1 -24939.057,E2 -24939.057} C_VEL
LIN {X 0,Y 134.851,Z 380.816,A -85,B 0,C 180,E1 -24943.568,E2 -24943.568} C_VEL
LIN {X 0,Y 136.405,Z 376.672,A -85,B 0,C 180,E1 -24948.012,E2 -24948.012} C_VEL
LIN {X 0,Y 139.226,Z 370.331,A -85,B 0,C 180,E1 -24953.034,E2 -24953.034} C_VEL
LIN {X 0,Y 141.26,Z 365.926,A -85,B 0,C 180,E1 -24955.811,E2 -24955.811} C_VEL
LIN {X 0,Y 144.249,Z 359.39,A -85,B 0,C 180,E1 -24959.162,E2 -24959.162} C_VEL
LIN {X 0,Y 147.628,Z 351.528,A -85,B 0,C 180,E1 -24962.387,E2 -24962.387} C_VEL
LIN {X 0,Y 149.561,Z 342.904,A -85,B 0,C 180,E1 -24965.529,E2 -24965.529} C_VEL
LIN {X 0,Y 150.926,Z 333.398,A -85,B 0,C 180,E1 -24968.525,E2 -24968.525} C_VEL
LIN {X 0,Y 151.566,Z 322.622,A -85,B 0,C 180,E1 -24971.527,E2 -24971.527} C_VEL
LIN {X 0,Y 151.229,Z 311.545,A -85,B 0,C 180,E1 -24974.35,E2 -24974.35} C_VEL
LIN {X 0,Y 150.533,Z 307.053,A -85,B 0,C 180,E1 -24975.548,E2 -24975.548} C_VEL
LIN {X 0,Y 147.594,Z 298.894,A -85,B 0,C 180,E1 -24978.192,E2 -24978.192} C_VEL
LIN {X 0,Y 145.243,Z 293.822,A -85,B 0,C 180,E1 -24980.01,E2 -24980.01} C_VEL
LIN {X 0,Y 143.165,Z 289.411,A -85,B 0,C 180,E1 -24981.614,E2 -24981.614} C_VEL
LIN {X 0,Y 141.086,Z 285.527,A -85,B 0,C 180,E1 -24983.168,E2 -24983.168} C_VEL
LIN {X 0,Y 140.457,Z 284.109,A -85,B 0,C 180,E1 -24983.659,E2 -24983.659} C_VEL
LIN {X 0,Y 139.461,Z 283.022,A -85,B 0,C 180,E1 -24984.304,E2 -24984.304} C_VEL
LIN {X 0,Y 135.447,Z 279.952,A -85,B 0,C 180,E1 -24986.944,E2 -24986.944} C_VEL
LIN {X 0,Y 130.716,Z 277.808,A -85,B 0,C 180,E1 -24990.313,E2 -24990.313} C_VEL
LIN {X 0,Y 129.803,Z 277.084,A -85,B 0,C 180,E1 -24991.968,E2 -24991.968} C_VEL
LIN {X 0,Y 129.581,Z 274.827,A -85,B 0,C 180,E1 -24997.688,E2 -24997.688} C_VEL
LIN {X 0,Y 129.389,Z 273.729,A -85,B 0,C 180,E1 -25000.98,E2 -25000.98} C_VEL
LIN {X 0,Y 129.215,Z 272.757,A -85,B 0,C 180,E1 -25004.22,E2 -25004.22} C_VEL
LIN {X 0,Y 129.353,Z 272.375,A -85,B 0,C 180,E1 -25007.973,E2 -25007.973} C_VEL
LIN {X 0,Y 129.48,Z 272.36,A -85,B 0,C 180,E1 -25010.629,E2 -25010.629} C_VEL
LIN {X 0,Y 130.083,Z 272.275,A -85,B 0,C 180,E1 -25020,E2 -25020} C_VEL
LIN {X 0,Y 129.471,Z 272.349,A -85,B 0,C 180,E1 -25029.373,E2 -25029.373} C_VEL
LIN {X 0,Y 129.308,Z 272.379,A -85,B 0,C 180,E1 -25032.557,E2 -25032.557} C_VEL
LIN {X 0,Y 129.093,Z 272.397,A -85,B 0,C 180,E1 -25039.066,E2 -25039.066} C_VEL
LIN {X 0,Y 129.044,Z 272.412,A -85,B 0,C 180,E1 -25042.411,E2 -25042.411} C_VEL
LIN {X 0,Y 129.008,Z 272.408,A -85,B 0,C 180,E1 -25049.361,E2 -25049.361} C_VEL
LIN {X 0,Y 128.998,Z 272.56,A -85,B 0,C 180,E1 -25053.366,E2 -25053.366} C_VEL
LIN {X 0,Y 129.958,Z 275.166,A -85,B 0,C 180,E1 -25054.504,E2 -25054.504} C_VEL
LIN {X 0,Y 131.802,Z 277.221,A -85,B 0,C 180,E1 -25056.149,E2 -25056.149} C_VEL
LIN {X 0,Y 132.726,Z 278.096,A -85,B 0,C 180,E1 -25056.92,E2 -25056.92} C_VEL
LIN {X 0,Y 134.345,Z 281.131,A -85,B 0,C 180,E1 -25058.482,E2 -25058.482} C_VEL
LIN {X 0,Y 135.894,Z 283.082,A -85,B 0,C 180,E1 -25059.792,E2 -25059.792} C_VEL
LIN {X 0,Y 140.938,Z 291.794,A -85,B 0,C 180,E1 -25064.277,E2 -25064.277} C_VEL
LIN {X 0,Y 144.665,Z 299.476,A -85,B 0,C 180,E1 -25067.806,E2 -25067.806} C_VEL
LIN {X 0,Y 146.892,Z 305.898,A -85,B 0,C 180,E1 -25070.41,E2 -25070.41} C_VEL
LIN {X 0,Y 148.338,Z 314.811,A -85,B 0,C 180,E1 -25073.653,E2 -25073.653} C_VEL
LIN {X 0,Y 148.624,Z 324.119,A -85,B 0,C 180,E1 -25077.053,E2 -25077.053} C_VEL
LIN {X 0,Y 148.055,Z 326.208,A -85,B 0,C 180,E1 -25077.718,E2 -25077.718} C_VEL
LIN {X 0,Y 143.999,Z 335.765,A -85,B 0,C 180,E1 -25080.782,E2 -25080.782} C_VEL
LIN {X 0,Y 140.347,Z 343.593,A -85,B 0,C 180,E1 -25084.009,E2 -25084.009} C_VEL
LIN {X 0,Y 136.612,Z 351.299,A -85,B 0,C 180,E1 -25088.141,E2 -25088.141} C_VEL
LIN {X 0,Y 132.909,Z 358.272,A -85,B 0,C 180,E1 -25093.088,E2 -25093.088} C_VEL
LIN {X 0,Y 130.324,Z 362.971,A -85,B 0,C 180,E1 -25097.538,E2 -25097.538} C_VEL
LIN {X 0,Y 128.58,Z 366.562,A -85,B 0,C 180,E1 -25102.142,E2 -25102.142} C_VEL
LIN {X 0,Y 127.506,Z 369.158,A -85,B 0,C 180,E1 -25106.836,E2 -25106.836} C_VEL
LIN {X 0,Y 127.177,Z 370.383,A -85,B 0,C 180,E1 -25109.995,E2 -25109.995} C_VEL
LIN {X 0,Y 127.127,Z 371.58,A -85,B 0,C 180,E1 -25115.67,E2 -25115.67} C_VEL
LIN {X 0,Y 127.483,Z 371.657,A -85,B 0,C 180,E1 -25119.515,E2 -25119.515} C_VEL
LIN {X 0,Y 128.027,Z 371.321,A -85,B 0,C 180,E1 -25122.679,E2 -25122.679} C_VEL
LIN {X 0,Y 128.89,Z 370.588,A -85,B 0,C 180,E1 -25125.816,E2 -25125.816} C_VEL
LIN {X 0,Y 131.576,Z 367.847,A -85,B 0,C 180,E1 -25131.951,E2 -25131.951} C_VEL
LIN {X 0,Y 134.496,Z 364.666,A -85,B 0,C 180,E1 -25136.365,E2 -25136.365} C_VEL
LIN {X 0,Y 138.034,Z 360.417,A -85,B 0,C 180,E1 -25140.602,E2 -25140.602} C_VEL
LIN {X 0,Y 142.271,Z 354.967,A -85,B 0,C 180,E1 -25144.611,E2 -25144.611} C_VEL
LIN {X 0,Y 147.049,Z 348.14,A -85,B 0,C 180,E1 -25148.407,E2 -25148.407} C_VEL
LIN {X 0,Y 152.232,Z 339.804,A -85,B 0,C 180,E1 -25151.88,E2 -25151.88} C_VEL
LIN {X 0,Y 155.13,Z 334.479,A -85,B 0,C 180,E1 -25153.693,E2 -25153.693} C_VEL
LIN {X 0,Y 155.539,Z 327.66,A -85,B 0,C 180,E1 -25156.811,E2 -25156.811} C_VEL
LIN {X 0,Y 155.135,Z 321.213,A -85,B 0,C 180,E1 -25159.793,E2 -25159.793} C_VEL
LIN {X 0,Y 153.523,Z 313.874,A -85,B 0,C 180,E1 -25163.479,E2 -25163.479} C_VEL
LIN {X 0,Y 151.809,Z 308.446,A -85,B 0,C 180,E1 -25166.433,E2 -25166.433} C_VEL
LIN {X 0,Y 149.222,Z 301.943,A -85,B 0,C 180,E1 -25170.361,E2 -25170.361} C_VEL
LIN {X 0,Y 146.963,Z 297.698,A -85,B 0,C 180,E1 -25173.452,E2 -25173.452} C_VEL
LIN {X 0,Y 145.396,Z 294.674,A -85,B 0,C 180,E1 -25175.74,E2 -25175.74} C_VEL
LIN {X 0,Y 142.72,Z 290.188,A -85,B 0,C 180,E1 -25179.836,E2 -25179.836} C_VEL
LIN {X 0,Y 139.783,Z 286.231,A -85,B 0,C 180,E1 -25184.881,E2 -25184.881} C_VEL
LIN {X 0,Y 139.335,Z 284.85,A -85,B 0,C 180,E1 -25186.137,E2 -25186.137} C_VEL
LIN {X 0,Y 135.867,Z 280.943,A -85,B 0,C 180,E1 -25196.849,E2 -25196.849} C_VEL
LIN {X 0,Y 135.788,Z 280.208,A -85,B 0,C 180,E1 -25198.517,E2 -25198.517} C_VEL
LIN {X 0,Y 135.732,Z 281.273,A -85,B 0,C 180,E1 -25205.571,E2 -25205.571} C_VEL
LIN {X 0,Y 136.557,Z 284.584,A -85,B 0,C 180,E1 -25211.127,E2 -25211.127} C_VEL
LIN {X 0,Y 139.526,Z 289.193,A -85,B 0,C 180,E1 -25218.349,E2 -25218.349} C_VEL
LIN {X 0,Y 139.943,Z 290.131,A -85,B 0,C 180,E1 -25219.252,E2 -25219.252} C_VEL
LIN {X 0,Y 141.235,Z 293.449,A -85,B 0,C 180,E1 -25221.913,E2 -25221.913} C_VEL
LIN {X 0,Y 143.089,Z 296.194,A -85,B 0,C 180,E1 -25224.676,E2 -25224.676} C_VEL
LIN {X 0,Y 144.785,Z 300.424,A -85,B 0,C 180,E1 -25227.46,E2 -25227.46} C_VEL
LIN {X 0,Y 145.794,Z 302.215,A -85,B 0,C 180,E1 -25228.819,E2 -25228.819} C_VEL
LIN {X 0,Y 148.533,Z 309.477,A -85,B 0,C 180,E1 -25232.965,E2 -25232.965} C_VEL
LIN {X 0,Y 150.884,Z 316.103,A -85,B 0,C 180,E1 -25236.433,E2 -25236.433} C_VEL
LIN {X 0,Y 152.951,Z 323.831,A -85,B 0,C 180,E1 -25240.037,E2 -25240.037} C_VEL
LIN {X 0,Y 153.446,Z 326.67,A -85,B 0,C 180,E1 -25241.255,E2 -25241.255} C_VEL
LIN {X 0,Y 152.637,Z 336.192,A -85,B 0,C 180,E1 -25244.547,E2 -25244.547} C_VEL
LIN {X 0,Y 150.804,Z 345.461,A -85,B 0,C 180,E1 -25247.91,E2 -25247.91} C_VEL
LIN {X 0,Y 148.574,Z 353.483,A -85,B 0,C 180,E1 -25251.193,E2 -25251.193} C_VEL
LIN {X 0,Y 146.443,Z 358.089,A -85,B 0,C 180,E1 -25253.143,E2 -25253.143} C_VEL
LIN {X 0,Y 141.383,Z 365.839,A -85,B 0,C 180,E1 -25256.858,E2 -25256.858} C_VEL
LIN {X 0,Y 137.055,Z 372.094,A -85,B 0,C 180,E1 -25260.858,E2 -25260.858} C_VEL
LIN {X 0,Y 133.421,Z 377.076,A -85,B 0,C 180,E1 -25265.082,E2 -25265.082} C_VEL
LIN {X 0,Y 130.517,Z 380.949,A -85,B 0,C 180,E1 -25269.517,E2 -25269.517} C_VEL
LIN {X 0,Y 128.421,Z 383.814,A -85,B 0,C 180,E1 -25274.124,E2 -25274.124} C_VEL
LIN {X 0,Y 126.927,Z 386.171,A -85,B 0,C 180,E1 -25280.443,E2 -25280.443} C_VEL
LIN {X 0,Y 126.694,Z 386.765,A -85,B 0,C 180,E1 -25283.635,E2 -25283.635} C_VEL
LIN {X 0,Y 126.698,Z 386.923,A -85,B 0,C 180,E1 -25286.825,E2 -25286.825} C_VEL
LIN {X 0,Y 126.918,Z 386.682,A -85,B 0,C 180,E1 -25290.005,E2 -25290.005} C_VEL
LIN {X 0,Y 126.746,Z 385.919,A -85,B 0,C 180,E1 -25293.541,E2 -25293.541} C_VEL
LIN {X 0,Y 126.754,Z 384.936,A -85,B 0,C 180,E1 -25296.371,E2 -25296.371} C_VEL
LIN {X 0,Y 126.958,Z 383.398,A -85,B 0,C 180,E1 -25299.564,E2 -25299.564} C_VEL
LIN {X 0,Y 127.933,Z 380.297,A -85,B 0,C 180,E1 -25304.317,E2 -25304.317} C_VEL
LIN {X 0,Y 129.636,Z 376.125,A -85,B 0,C 180,E1 -25308.987,E2 -25308.987} C_VEL
LIN {X 0,Y 132.685,Z 369.755,A -85,B 0,C 180,E1 -25314.241,E2 -25314.241} C_VEL
LIN {X 0,Y 134.759,Z 365.312,A -85,B 0,C 180,E1 -25317.155,E2 -25317.155} C_VEL
LIN {X 0,Y 138.743,Z 357.259,A -85,B 0,C 180,E1 -25321.284,E2 -25321.284} C_VEL
LIN {X 0,Y 141.497,Z 350.827,A -85,B 0,C 180,E1 -25323.976,E2 -25323.976} C_VEL
LIN {X 0,Y 143.564,Z 341.71,A -85,B 0,C 180,E1 -25327.421,E2 -25327.421} C_VEL
LIN {X 0,Y 145.077,Z 331.165,A -85,B 0,C 180,E1 -25330.848,E2 -25330.848} C_VEL
LIN {X 0,Y 145.662,Z 321.554,A -85,B 0,C 180,E1 -25333.637,E2 -25333.637} C_VEL
LIN {X 0,Y 145.499,Z 312.503,A -85,B 0,C 180,E1 -25336.099,E2 -25336.099} C_VEL
LIN {X 0,Y 143.4,Z 305.256,A -85,B 0,C 180,E1 -25338.576,E2 -25338.576} C_VEL
LIN {X 0,Y 141.153,Z 299.306,A -85,B 0,C 180,E1 -25340.781,E2 -25340.781} C_VEL
LIN {X 0,Y 138.542,Z 293.779,A -85,B 0,C 180,E1 -25343.072,E2 -25343.072} C_VEL
LIN {X 0,Y 136.36,Z 289.224,A -85,B 0,C 180,E1 -25345.014,E2 -25345.014} C_VEL
LIN {X 0,Y 134.1,Z 285.271,A -85,B 0,C 180,E1 -25346.955,E2 -25346.955} C_VEL
LIN {X 0,Y 133.424,Z 283.664,A -85,B 0,C 180,E1 -25347.603,E2 -25347.603} C_VEL
LIN {X 0,Y 130.96,Z 280.534,A -85,B 0,C 180,E1 -25349.643,E2 -25349.643} C_VEL
LIN {X 0,Y 129.942,Z 277.528,A -85,B 0,C 180,E1 -25350.872,E2 -25350.872} C_VEL
LIN {X 0,Y 129.803,Z 277.084,A -85,B 0,C 180,E1 -25351.968,E2 -25351.968} C_VEL
LIN {X 0,Y 128.91,Z 276.218,A -85,B 0,C 180,E1 -25354.522,E2 -25354.522} C_VEL
LIN {X 0,Y 127.179,Z 275.622,A -85,B 0,C 180,E1 -25357.055,E2 -25357.055} C_VEL
LIN {X 0,Y 122.537,Z 274.386,A -85,B 0,C 180,E1 -25364.096,E2 -25364.096} C_VEL
LIN {X 0,Y 122.252,Z 273.94,A -85,B 0,C 180,E1 -25365.958,E2 -25365.958} C_VEL
LIN {X 0,Y 122.406,Z 273.24,A -85,B 0,C 180,E1 -25370.082,E2 -25370.082} C_VEL
LIN {X 0,Y 122.604,Z 273.207,A -85,B 0,C 180,E1 -25376.714,E2 -25376.714} C_VEL
LIN {X 0,Y 123.035,Z 273.152,A -85,B 0,C 180,E1 -25380,E2 -25380} C_VEL
LIN {X 0,Y 122.398,Z 273.234,A -85,B 0,C 180,E1 -25386.87,E2 -25386.87} C_VEL
LIN {X 0,Y 122.297,Z 273.252,A -85,B 0,C 180,E1 -25392.309,E2 -25392.309} C_VEL
LIN {X 0,Y 122.073,Z 273.278,A -85,B 0,C 180,E1 -25396.73,E2 -25396.73} C_VEL
LIN {X 0,Y 121.988,Z 273.288,A -85,B 0,C 180,E1 -25402.799,E2 -25402.799} C_VEL
LIN {X 0,Y 121.934,Z 273.497,A -85,B 0,C 180,E1 -25407.343,E2 -25407.343} C_VEL
LIN {X 0,Y 122.702,Z 275.769,A -85,B 0,C 180,E1 -25408.595,E2 -25408.595} C_VEL
LIN {X 0,Y 124.878,Z 278.237,A -85,B 0,C 180,E1 -25411.136,E2 -25411.136} C_VEL
LIN {X 0,Y 125.982,Z 279.019,A -85,B 0,C 180,E1 -25412.239,E2 -25412.239} C_VEL
LIN {X 0,Y 127.522,Z 282.059,A -85,B 0,C 180,E1 -25414.11,E2 -25414.11} C_VEL
LIN {X 0,Y 129.296,Z 284.052,A -85,B 0,C 180,E1 -25415.875,E2 -25415.875} C_VEL
LIN {X 0,Y 131.022,Z 287.174,A -85,B 0,C 180,E1 -25417.753,E2 -25417.753} C_VEL
LIN {X 0,Y 131.939,Z 288.339,A -85,B 0,C 180,E1 -25418.629,E2 -25418.629} C_VEL
LIN {X 0,Y 136.404,Z 296.683,A -85,B 0,C 180,E1 -25423.283,E2 -25423.283} C_VEL
LIN {X 0,Y 140.144,Z 305.335,A -85,B 0,C 180,E1 -25427.55,E2 -25427.55} C_VEL
LIN {X 0,Y 141.544,Z 310.594,A -85,B 0,C 180,E1 -25429.793,E2 -25429.793} C_VEL
LIN {X 0,Y 142.52,Z 319.444,A -85,B 0,C 180,E1 -25433.288,E2 -25433.288} C_VEL
LIN {X 0,Y 142.437,Z 325.934,A -85,B 0,C 180,E1 -25435.853,E2 -25435.853} C_VEL
LIN {X 0,Y 138.717,Z 334.706,A -85,B 0,C 180,E1 -25438.709,E2 -25438.709} C_VEL
LIN {X 0,Y 134.048,Z 344.253,A -85,B 0,C 180,E1 -25442.689,E2 -25442.689} C_VEL
LIN {X 0,Y 130.38,Z 351.353,A -85,B 0,C 180,E1 -25446.62,E2 -25446.62} C_VEL
LIN {X 0,Y 127.169,Z 357.049,A -85,B 0,C 180,E1 -25450.63,E2 -25450.63} C_VEL
LIN {X 0,Y 124.273,Z 362.096,A -85,B 0,C 180,E1 -25455.252,E2 -25455.252} C_VEL
LIN {X 0,Y 122.115,Z 366.018,A -85,B 0,C 180,E1 -25460.053,E2 -25460.053} C_VEL
LIN {X 0,Y 121.104,Z 368.035,A -85,B 0,C 180,E1 -25463.33,E2 -25463.33} C_VEL
LIN {X 0,Y 120.456,Z 369.641,A -85,B 0,C 180,E1 -25466.65,E2 -25466.65} C_VEL
LIN {X 0,Y 120.093,Z 370.854,A -85,B 0,C 180,E1 -25469.995,E2 -25469.995} C_VEL
LIN {X 0,Y 120.065,Z 371.988,A -85,B 0,C 180,E1 -25475.671,E2 -25475.671} C_VEL
LIN {X 0,Y 120.46,Z 372.08,A -85,B 0,C 180,E1 -25480.075,E2 -25480.075} C_VEL
LIN {X 0,Y 121.096,Z 371.73,A -85,B 0,C 180,E1 -25483.418,E2 -25483.418} C_VEL
LIN {X 0,Y 122.056,Z 370.972,A -85,B 0,C 180,E1 -25486.727,E2 -25486.727} C_VEL
LIN {X 0,Y 124.998,Z 368.204,A -85,B 0,C 180,E1 -25493.172,E2 -25493.172} C_VEL
LIN {X 0,Y 128.12,Z 364.997,A -85,B 0,C 180,E1 -25497.787,E2 -25497.787} C_VEL
LIN {X 0,Y 131.95,Z 360.716,A -85,B 0,C 180,E1 -25502.178,E2 -25502.178} C_VEL
LIN {X 0,Y 136.463,Z 355.234,A -85,B 0,C 180,E1 -25506.312,E2 -25506.312} C_VEL
LIN {X 0,Y 141.526,Z 348.368,A -85,B 0,C 180,E1 -25510.202,E2 -25510.202} C_VEL
LIN {X 0,Y 146.816,Z 340.251,A -85,B 0,C 180,E1 -25513.642,E2 -25513.642} C_VEL
LIN {X 0,Y 149.067,Z 336.396,A -85,B 0,C 180,E1 -25515.001,E2 -25515.001} C_VEL
LIN {X 0,Y 149.677,Z 330.792,A -85,B 0,C 180,E1 -25517.742,E2 -25517.742} C_VEL
LIN {X 0,Y 149.479,Z 323.936,A -85,B 0,C 180,E1 -25521.191,E2 -25521.191} C_VEL
LIN {X 0,Y 148.042,Z 316.612,A -85,B 0,C 180,E1 -25525.272,E2 -25525.272} C_VEL
LIN {X 0,Y 146.193,Z 310.576,A -85,B 0,C 180,E1 -25528.963,E2 -25528.963} C_VEL
LIN {X 0,Y 144.235,Z 305.583,A -85,B 0,C 180,E1 -25532.425,E2 -25532.425} C_VEL
LIN {X 0,Y 141.777,Z 300.427,A -85,B 0,C 180,E1 -25536.636,E2 -25536.636} C_VEL
LIN {X 0,Y 139.471,Z 296.119,A -85,B 0,C 180,E1 -25540.88,E2 -25540.88} C_VEL
LIN {X 0,Y 136.233,Z 291.029,A -85,B 0,C 180,E1 -25548.091,E2 -25548.091} C_VEL
LIN {X 0,Y 134.037,Z 287.571,A -85,B 0,C 180,E1 -25557.558,E2 -25557.558} C_VEL
LIN {X 0,Y 134.05,Z 287.102,A -85,B 0,C 180,E1 -25558.498,E2 -25558.498} C_VEL
LIN {X 0,Y 133.932,Z 288.043,A -85,B 0,C 180,E1 -25565.034,E2 -25565.034} C_VEL
LIN {X 0,Y 134.41,Z 290.822,A -85,B 0,C 180,E1 -25569.974,E2 -25569.974} C_VEL
LIN {X 0,Y 137.104,Z 295.783,A -85,B 0,C 180,E1 -25577.912,E2 -25577.912} C_VEL
LIN {X 0,Y 138.177,Z 299.368,A -85,B 0,C 180,E1 -25580.857,E2 -25580.857} C_VEL
LIN {X 0,Y 139.795,Z 302.052,A -85,B 0,C 180,E1 -25583.715,E2 -25583.715} C_VEL
LIN {X 0,Y 141.212,Z 306.18,A -85,B 0,C 180,E1 -25586.61,E2 -25586.61} C_VEL
LIN {X 0,Y 142.068,Z 308.027,A -85,B 0,C 180,E1 -25588.031,E2 -25588.031} C_VEL
LIN {X 0,Y 144.825,Z 316.357,A -85,B 0,C 180,E1 -25593.089,E2 -25593.089} C_VEL
LIN {X 0,Y 147.052,Z 324.64,A -85,B 0,C 180,E1 -25597.543,E2 -25597.543} C_VEL
LIN {X 0,Y 147.9,Z 329.688,A -85,B 0,C 180,E1 -25599.963,E2 -25599.963} C_VEL
LIN {X 0,Y 147.199,Z 336.098,A -85,B 0,C 180,E1 -25602.354,E2 -25602.354} C_VEL
LIN {X 0,Y 145.507,Z 344.402,A -85,B 0,C 180,E1 -25605.553,E2 -25605.553} C_VEL
LIN {X 0,Y 142.845,Z 353.281,A -85,B 0,C 180,E1 -25609.321,E2 -25609.321} C_VEL
LIN {X 0,Y 140.774,Z 357.87,A -85,B 0,C 180,E1 -25611.393,E2 -25611.393} C_VEL
LIN {X 0,Y 135.46,Z 365.571,A -85,B 0,C 180,E1 -25615.206,E2 -25615.206} C_VEL
LIN {X 0,Y 130.461,Z 372.31,A -85,B 0,C 180,E1 -25619.734,E2 -25619.734} C_VEL
LIN {X 0,Y 126.993,Z 376.749,A -85,B 0,C 180,E1 -25623.727,E2 -25623.727} C_VEL
LIN {X 0,Y 123.871,Z 380.597,A -85,B 0,C 180,E1 -25628.364,E2 -25628.364} C_VEL
LIN {X 0,Y 121.554,Z 383.435,A -85,B 0,C 180,E1 -25633.202,E2 -25633.202} C_VEL
LIN {X 0,Y 119.919,Z 385.772,A -85,B 0,C 180,E1 -25639.879,E2 -25639.879} C_VEL
LIN {X 0,Y 119.632,Z 386.348,A -85,B 0,C 180,E1 -25643.258,E2 -25643.258} C_VEL
LIN {X 0,Y 119.617,Z 386.468,A -85,B 0,C 180,E1 -25647.21,E2 -25647.21} C_VEL
LIN {X 0,Y 119.838,Z 386.238,A -85,B 0,C 180,E1 -25650.005,E2 -25650.005} C_VEL
LIN {X 0,Y 119.683,Z 385.556,A -85,B 0,C 180,E1 -25653.371,E2 -25653.371} C_VEL
LIN {X 0,Y 119.674,Z 384.462,A -85,B 0,C 180,E1 -25656.75,E2 -25656.75} C_VEL
LIN {X 0,Y 119.945,Z 382.905,A -85,B 0,C 180,E1 -25660.129,E2 -25660.129} C_VEL
LIN {X 0,Y 121.022,Z 379.776,A -85,B 0,C 180,E1 -25665.154,E2 -25665.154} C_VEL
LIN {X 0,Y 122.916,Z 375.579,A -85,B 0,C 180,E1 -25670.069,E2 -25670.069} C_VEL
LIN {X 0,Y 126.221,Z 369.18,A -85,B 0,C 180,E1 -25675.569,E2 -25675.569} C_VEL
LIN {X 0,Y 129.681,Z 362.332,A -85,B 0,C 180,E1 -25680.001,E2 -25680.001} C_VEL
LIN {X 0,Y 133.422,Z 355.107,A -85,B 0,C 180,E1 -25683.584,E2 -25683.584} C_VEL
LIN {X 0,Y 135.432,Z 350.115,A -85,B 0,C 180,E1 -25685.723,E2 -25685.723} C_VEL
LIN {X 0,Y 137.438,Z 341.625,A -85,B 0,C 180,E1 -25689.101,E2 -25689.101} C_VEL
LIN {X 0,Y 138.95,Z 333.001,A -85,B 0,C 180,E1 -25692.082,E2 -25692.082} C_VEL
LIN {X 0,Y 139.879,Z 322.643,A -85,B 0,C 180,E1 -25695.299,E2 -25695.299} C_VEL
LIN {X 0,Y 139.777,Z 314.475,A -85,B 0,C 180,E1 -25697.74,E2 -25697.74} C_VEL
LIN {X 0,Y 137.137,Z 305.913,A -85,B 0,C 180,E1 -25701.112,E2 -25701.112} C_VEL
LIN {X 0,Y 134.5,Z 299.217,A -85,B 0,C 180,E1 -25703.996,E2 -25703.996} C_VEL
LIN {X 0,Y 132.314,Z 294.359,A -85,B 0,C 180,E1 -25706.28,E2 -25706.28} C_VEL
LIN {X 0,Y 130.175,Z 289.956,A -85,B 0,C 180,E1 -25708.52,E2 -25708.52} C_VEL
LIN {X 0,Y 129.095,Z 288.351,A -85,B 0,C 180,E1 -25709.538,E2 -25709.538} C_VEL
LIN {X 0,Y 127.211,Z 284.966,A -85,B 0,C 180,E1 -25711.543,E2 -25711.543} C_VEL
LIN {X 0,Y 126.578,Z 283.347,A -85,B 0,C 180,E1 -25712.331,E2 -25712.331} C_VEL
LIN {X 0,Y 123.911,Z 280.096,A -85,B 0,C 180,E1 -25715.115,E2 -25715.115} C_VEL
LIN {X 0,Y 122.728,Z 277.065,A -85,B 0,C 180,E1 -25716.763,E2 -25716.763} C_VEL
LIN {X 0,Y 122.659,Z 276.632,A -85,B 0,C 180,E1 -25716.986,E2 -25716.986} C_VEL
LIN {X 0,Y 122.336,Z 274.659,A -85,B 0,C 180,E1 -25723.307,E2 -25723.307} C_VEL
LIN {X 0,Y 122.252,Z 273.94,A -85,B 0,C 180,E1 -25725.958,E2 -25725.958} C_VEL
LIN {X 0,Y 121.751,Z 273.5,A -85,B 0,C 180,E1 -25728.703,E2 -25728.703} C_VEL
LIN {X 0,Y 120.474,Z 273.494,A -85,B 0,C 180,E1 -25731.441,E2 -25731.441} C_VEL
LIN {X 0,Y 115.809,Z 274.048,A -85,B 0,C 180,E1 -25740.954,E2 -25740.954} C_VEL
LIN {X 0,Y 115.358,Z 274.116,A -85,B 0,C 180,E1 -25746.999,E2 -25746.999} C_VEL
LIN {X 0,Y 115.214,Z 274.133,A -85,B 0,C 180,E1 -25752.559,E2 -25752.559} C_VEL
LIN {X 0,Y 114.955,Z 274.288,A -85,B 0,C 180,E1 -25758.26,E2 -25758.26} C_VEL
LIN {X 0,Y 115.77,Z 276.669,A -85,B 0,C 180,E1 -25760.431,E2 -25760.431} C_VEL
LIN {X 0,Y 117.723,Z 279.003,A -85,B 0,C 180,E1 -25763.93,E2 -25763.93} C_VEL
LIN {X 0,Y 119.335,Z 280.15,A -85,B 0,C 180,E1 -25766.213,E2 -25766.213} C_VEL
LIN {X 0,Y 120.747,Z 283.034,A -85,B 0,C 180,E1 -25768.532,E2 -25768.532} C_VEL
LIN {X 0,Y 123.028,Z 285.555,A -85,B 0,C 180,E1 -25771.418,E2 -25771.418} C_VEL
LIN {X 0,Y 123.861,Z 287.335,A -85,B 0,C 180,E1 -25772.619,E2 -25772.619} C_VEL
LIN {X 0,Y 125.864,Z 290.144,A -85,B 0,C 180,E1 -25775.033,E2 -25775.033} C_VEL
LIN {X 0,Y 130.219,Z 298.239,A -85,B 0,C 180,E1 -25780.365,E2 -25780.365} C_VEL
LIN {X 0,Y 133.403,Z 305.459,A -85,B 0,C 180,E1 -25784.456,E2 -25784.456} C_VEL
LIN {X 0,Y 135.502,Z 311.624,A -85,B 0,C 180,E1 -25787.597,E2 -25787.597} C_VEL
LIN {X 0,Y 136.284,Z 316.918,A -85,B 0,C 180,E1 -25789.933,E2 -25789.933} C_VEL
LIN {X 0,Y 136.491,Z 324.704,A -85,B 0,C 180,E1 -25793.227,E2 -25793.227} C_VEL
LIN {X 0,Y 136.331,Z 327.739,A -85,B 0,C 180,E1 -25794.548,E2 -25794.548} C_VEL
LIN {X 0,Y 131.876,Z 337.179,A -85,B 0,C 180,E1 -25797.792,E2 -25797.792} C_VEL
LIN {X 0,Y 127.057,Z 346.255,A -85,B 0,C 180,E1 -25801.95,E2 -25801.95} C_VEL
LIN {X 0,Y 123.025,Z 353.545,A -85,B 0,C 180,E1 -25806.424,E2 -25806.424} C_VEL
LIN {X 0,Y 119.471,Z 359.41,A -85,B 0,C 180,E1 -25811.118,E2 -25811.118} C_VEL
LIN {X 0,Y 116.582,Z 364.048,A -85,B 0,C 180,E1 -25816.041,E2 -25816.041} C_VEL
LIN {X 0,Y 114.603,Z 367.583,A -85,B 0,C 180,E1 -25821.176,E2 -25821.176} C_VEL
LIN {X 0,Y 113.408,Z 370.124,A -85,B 0,C 180,E1 -25826.442,E2 -25826.442} C_VEL
LIN {X 0,Y 113.01,Z 371.325,A -85,B 0,C 180,E1 -25829.995,E2 -25829.995} C_VEL
LIN {X 0,Y 112.975,Z 372.371,A -85,B 0,C 180,E1 -25835.532,E2 -25835.532} C_VEL
LIN {X 0,Y 113.473,Z 372.501,A -85,B 0,C 180,E1 -25840.703,E2 -25840.703} C_VEL
LIN {X 0,Y 114.172,Z 372.14,A -85,B 0,C 180,E1 -25844.249,E2 -25844.249} C_VEL
LIN {X 0,Y 115.244,Z 371.357,A -85,B 0,C 180,E1 -25847.748,E2 -25847.748} C_VEL
LIN {X 0,Y 116.633,Z 370.162,A -85,B 0,C 180,E1 -25851.19,E2 -25851.19} C_VEL
LIN {X 0,Y 119.544,Z 367.594,A -85,B 0,C 180,E1 -25856.157,E2 -25856.157} C_VEL
LIN {X 0,Y 123.755,Z 363.384,A -85,B 0,C 180,E1 -25861.586,E2 -25861.586} C_VEL
LIN {X 0,Y 129.091,Z 357.503,A -85,B 0,C 180,E1 -25866.783,E2 -25866.783} C_VEL
LIN {X 0,Y 134.309,Z 351.052,A -85,B 0,C 180,E1 -25870.844,E2 -25870.844} C_VEL
LIN {X 0,Y 140.09,Z 343.004,A -85,B 0,C 180,E1 -25874.609,E2 -25874.609} C_VEL
LIN {X 0,Y 143.261,Z 337.829,A -85,B 0,C 180,E1 -25876.622,E2 -25876.622} C_VEL
LIN {X 0,Y 143.911,Z 332.461,A -85,B 0,C 180,E1 -25879.472,E2 -25879.472} C_VEL
LIN {X 0,Y 143.937,Z 327.878,A -85,B 0,C 180,E1 -25881.986,E2 -25881.986} C_VEL
LIN {X 0,Y 143.11,Z 321.859,A -85,B 0,C 180,E1 -25885.616,E2 -25885.616} C_VEL
LIN {X 0,Y 141.633,Z 315.781,A -85,B 0,C 180,E1 -25889.603,E2 -25889.603} C_VEL
LIN {X 0,Y 140.045,Z 311.027,A -85,B 0,C 180,E1 -25893.15,E2 -25893.15} C_VEL
LIN {X 0,Y 137.964,Z 306.043,A -85,B 0,C 180,E1 -25897.538,E2 -25897.538} C_VEL
LIN {X 0,Y 136.009,Z 301.948,A -85,B 0,C 180,E1 -25901.938,E2 -25901.938} C_VEL
LIN {X 0,Y 133.772,Z 297.981,A -85,B 0,C 180,E1 -25907.869,E2 -25907.869} C_VEL
LIN {X 0,Y 131.871,Z 294.702,A -85,B 0,C 180,E1 -25916.945,E2 -25916.945} C_VEL
LIN {X 0,Y 131.818,Z 293.934,A -85,B 0,C 180,E1 -25920,E2 -25920} C_VEL
LIN {X 0,Y 131.708,Z 294.444,A -85,B 0,C 180,E1 -25923.058,E2 -25923.058} C_VEL
LIN {X 0,Y 131.813,Z 295.43,A -85,B 0,C 180,E1 -25926.121,E2 -25926.121} C_VEL
LIN {X 0,Y 134.013,Z 301.831,A -85,B 0,C 180,E1 -25936.764,E2 -25936.764} C_VEL
LIN {X 0,Y 135.509,Z 306.494,A -85,B 0,C 180,E1 -25941.287,E2 -25941.287} C_VEL
LIN {X 0,Y 136.25,Z 307.818,A -85,B 0,C 180,E1 -25942.759,E2 -25942.759} C_VEL
LIN {X 0,Y 138.384,Z 314.887,A -85,B 0,C 180,E1 -25948.019,E2 -25948.019} C_VEL
LIN {X 0,Y 140.039,Z 320.607,A -85,B 0,C 180,E1 -25951.798,E2 -25951.798} C_VEL
LIN {X 0,Y 141.82,Z 328.643,A -85,B 0,C 180,E1 -25956.489,E2 -25956.489} C_VEL
LIN {X 0,Y 142.376,Z 333.032,A -85,B 0,C 180,E1 -25958.784,E2 -25958.784} C_VEL
LIN {X 0,Y 140.928,Z 341.275,A -85,B 0,C 180,E1 -25962.121,E2 -25962.121} C_VEL
LIN {X 0,Y 138.412,Z 349.71,A -85,B 0,C 180,E1 -25965.693,E2 -25965.693} C_VEL
LIN {X 0,Y 135.988,Z 356.157,A -85,B 0,C 180,E1 -25968.788,E2 -25968.788} C_VEL
LIN {X 0,Y 133.38,Z 360.379,A -85,B 0,C 180,E1 -25970.786,E2 -25970.786} C_VEL
LIN {X 0,Y 127.962,Z 367.543,A -85,B 0,C 180,E1 -25974.788,E2 -25974.788} C_VEL
LIN {X 0,Y 123.329,Z 373.285,A -85,B 0,C 180,E1 -25979.15,E2 -25979.15} C_VEL
LIN {X 0,Y 119.418,Z 377.832,A -85,B 0,C 180,E1 -25983.813,E2 -25983.813} C_VEL
LIN {X 0,Y 116.29,Z 381.31,A -85,B 0,C 180,E1 -25988.745,E2 -25988.745} C_VEL
LIN {X 0,Y 113.644,Z 384.41,A -85,B 0,C 180,E1 -25995.684,E2 -25995.684} C_VEL
LIN {X 0,Y 112.907,Z 385.371,A -85,B 0,C 180,E1 -25999.243,E2 -25999.243} C_VEL
LIN {X 0,Y 112.57,Z 385.927,A -85,B 0,C 180,E1 -26002.832,E2 -26002.832} C_VEL
LIN {X 0,Y 112.556,Z 386.02,A -85,B 0,C 180,E1 -26007.49,E2 -26007.49} C_VEL
LIN {X 0,Y 112.758,Z 385.794,A -85,B 0,C 180,E1 -26010.005,E2 -26010.005} C_VEL
LIN {X 0,Y 112.586,Z 385.098,A -85,B 0,C 180,E1 -26013.584,E2 -26013.584} C_VEL
LIN {X 0,Y 112.6,Z 383.984,A -85,B 0,C 180,E1 -26017.176,E2 -26017.176} C_VEL
LIN {X 0,Y 112.929,Z 382.41,A -85,B 0,C 180,E1 -26020.766,E2 -26020.766} C_VEL
LIN {X 0,Y 114.126,Z 379.254,A -85,B 0,C 180,E1 -26026.093,E2 -26026.093} C_VEL
LIN {X 0,Y 116.249,Z 375.033,A -85,B 0,C 180,E1 -26031.274,E2 -26031.274} C_VEL
LIN {X 0,Y 119.837,Z 368.606,A -85,B 0,C 180,E1 -26037.039,E2 -26037.039} C_VEL
LIN {X 0,Y 122.879,Z 362.843,A -85,B 0,C 180,E1 -26040.986,E2 -26040.986} C_VEL
LIN {X 0,Y 127.53,Z 354.459,A -85,B 0,C 180,E1 -26045.36,E2 -26045.36} C_VEL
LIN {X 0,Y 129.448,Z 349.394,A -85,B 0,C 180,E1 -26047.652,E2 -26047.652} C_VEL
LIN {X 0,Y 131.67,Z 340.711,A -85,B 0,C 180,E1 -26051.229,E2 -26051.229} C_VEL
LIN {X 0,Y 133.367,Z 331.391,A -85,B 0,C 180,E1 -26054.571,E2 -26054.571} C_VEL
LIN {X 0,Y 134.294,Z 321.068,A -85,B 0,C 180,E1 -26057.943,E2 -26057.943} C_VEL
LIN {X 0,Y 134.352,Z 318.319,A -85,B 0,C 180,E1 -26058.83,E2 -26058.83} C_VEL
LIN {X 0,Y 132.726,Z 311.656,A -85,B 0,C 180,E1 -26061.622,E2 -26061.622} C_VEL
LIN {X 0,Y 129.887,Z 303.647,A -85,B 0,C 180,E1 -26065.38,E2 -26065.38} C_VEL
LIN {X 0,Y 128.078,Z 299.212,A -85,B 0,C 180,E1 -26067.656,E2 -26067.656} C_VEL
LIN {X 0,Y 125.944,Z 294.49,A -85,B 0,C 180,E1 -26070.314,E2 -26070.314} C_VEL
LIN {X 0,Y 123.924,Z 290.659,A -85,B 0,C 180,E1 -26072.791,E2 -26072.791} C_VEL
LIN {X 0,Y 123.222,Z 289.05,A -85,B 0,C 180,E1 -26073.777,E2 -26073.777} C_VEL
LIN {X 0,Y 120.769,Z 285.326,A -85,B 0,C 180,E1 -26076.885,E2 -26076.885} C_VEL
LIN {X 0,Y 119.856,Z 282.737,A -85,B 0,C 180,E1 -26078.475,E2 -26078.475} C_VEL
LIN {X 0,Y 116.825,Z 279.289,A -85,B 0,C 180,E1 -26082.946,E2 -26082.946} C_VEL
LIN {X 0,Y 115.434,Z 275.936,A -85,B 0,C 180,E1 -26085.977,E2 -26085.977} C_VEL
LIN {X 0,Y 115.375,Z 275.476,A -85,B 0,C 180,E1 -26086.473,E2 -26086.473} C_VEL
LIN {X 0,Y 115.409,Z 274.748,A -85,B 0,C 180,E1 -26089.474,E2 -26089.474} C_VEL
LIN {X 0,Y 115.371,Z 274.11,A -85,B 0,C 180,E1 -26093.002,E2 -26093.002} C_VEL
LIN {X 0,Y 115.986,Z 274.03,A -85,B 0,C 180,E1 -26100,E2 -26100} C_VEL
LIN {X 0,Y 115.809,Z 274.048,A -85,B 0,C 180,E1 -26100.954,E2 -26100.954} C_VEL
LIN {X 0,Y 115,Z 274.635,A -85,B 0,C 180,E1 -26103.847,E2 -26103.847} C_VEL
LIN {X 0,Y 113.071,Z 277.1,A -85,B 0,C 180,E1 -26108.585,E2 -26108.585} C_VEL
LIN {X 0,Y 112.06,Z 279.35,A -85,B 0,C 180,E1 -26112.453,E2 -26112.453} C_VEL
LIN {X 0,Y 112.261,Z 280.585,A -85,B 0,C 180,E1 -26115.422,E2 -26115.422} C_VEL
LIN {X 0,Y 112.596,Z 280.827,A -85,B 0,C 180,E1 -26116.41,E2 -26116.41} C_VEL
LIN {X 0,Y 112.955,Z 281.135,A -85,B 0,C 180,E1 -26117.307,E2 -26117.307} C_VEL
LIN {X 0,Y 114.223,Z 284.286,A -85,B 0,C 180,E1 -26120.956,E2 -26120.956} C_VEL
LIN {X 0,Y 116.65,Z 286.669,A -85,B 0,C 180,E1 -26125.283,E2 -26125.283} C_VEL
LIN {X 0,Y 118.309,Z 289.899,A -85,B 0,C 180,E1 -26128.375,E2 -26128.375} C_VEL
LIN {X 0,Y 119.241,Z 290.912,A -85,B 0,C 180,E1 -26129.693,E2 -26129.693} C_VEL
LIN {X 0,Y 122.2,Z 295.891,A -85,B 0,C 180,E1 -26134.108,E2 -26134.108} C_VEL
LIN {X 0,Y 125.549,Z 302.817,A -85,B 0,C 180,E1 -26139.033,E2 -26139.033} C_VEL
LIN {X 0,Y 128.205,Z 309.368,A -85,B 0,C 180,E1 -26143.142,E2 -26143.142} C_VEL
LIN {X 0,Y 130.154,Z 315.954,A -85,B 0,C 180,E1 -26146.798,E2 -26146.798} C_VEL
LIN {X 0,Y 130.599,Z 322.28,A -85,B 0,C 180,E1 -26149.772,E2 -26149.772} C_VEL
LIN {X 0,Y 130.345,Z 328.661,A -85,B 0,C 180,E1 -26152.71,E2 -26152.71} C_VEL
LIN {X 0,Y 127.822,Z 334.351,A -85,B 0,C 180,E1 -26154.732,E2 -26154.732} C_VEL
LIN {X 0,Y 123.331,Z 342.632,A -85,B 0,C 180,E1 -26158.184,E2 -26158.184} C_VEL
LIN {X 0,Y 119.299,Z 349.507,A -85,B 0,C 180,E1 -26161.877,E2 -26161.877} C_VEL
LIN {X 0,Y 115.246,Z 356.229,A -85,B 0,C 180,E1 -26166.642,E2 -26166.642} C_VEL
LIN {X 0,Y 111.711,Z 361.625,A -85,B 0,C 180,E1 -26171.66,E2 -26171.66} C_VEL
LIN {X 0,Y 108.979,Z 365.851,A -85,B 0,C 180,E1 -26176.95,E2 -26176.95} C_VEL
LIN {X 0,Y 107.093,Z 369.027,A -85,B 0,C 180,E1 -26182.453,E2 -26182.453} C_VEL
LIN {X 0,Y 106.363,Z 370.606,A -85,B 0,C 180,E1 -26186.206,E2 -26186.206} C_VEL
LIN {X 0,Y 105.929,Z 371.793,A -85,B 0,C 180,E1 -26189.994,E2 -26189.994} C_VEL
LIN {X 0,Y 105.87,Z 372.737,A -85,B 0,C 180,E1 -26195.277,E2 -26195.277} C_VEL
LIN {X 0,Y 106.471,Z 372.924,A -85,B 0,C 180,E1 -26201.416,E2 -26201.416} C_VEL
LIN {X 0,Y 107.288,Z 372.548,A -85,B 0,C 180,E1 -26205.184,E2 -26205.184} C_VEL
LIN {X 0,Y 108.456,Z 371.742,A -85,B 0,C 180,E1 -26208.899,E2 -26208.899} C_VEL
LIN {X 0,Y 110.006,Z 370.534,A -85,B 0,C 180,E1 -26212.534,E2 -26212.534} C_VEL
LIN {X 0,Y 113.183,Z 367.939,A -85,B 0,C 180,E1 -26217.75,E2 -26217.75} C_VEL
LIN {X 0,Y 117.394,Z 364.017,A -85,B 0,C 180,E1 -26223.055,E2 -26223.055} C_VEL
LIN {X 0,Y 121.725,Z 359.603,A -85,B 0,C 180,E1 -26227.311,E2 -26227.311} C_VEL
LIN {X 0,Y 127.072,Z 353.602,A -85,B 0,C 180,E1 -26231.575,E2 -26231.575} C_VEL
LIN {X 0,Y 133.008,Z 346.114,A -85,B 0,C 180,E1 -26235.499,E2 -26235.499} C_VEL
LIN {X 0,Y 136.686,Z 340.808,A -85,B 0,C 180,E1 -26237.695,E2 -26237.695} C_VEL
LIN {X 0,Y 137.465,Z 339.32,A -85,B 0,C 180,E1 -26238.345,E2 -26238.345} C_VEL
LIN {X 0,Y 138.233,Z 333.568,A -85,B 0,C 180,E1 -26241.716,E2 -26241.716} C_VEL
LIN {X 0,Y 138.164,Z 329.161,A -85,B 0,C 180,E1 -26244.468,E2 -26244.468} C_VEL
LIN {X 0,Y 137.411,Z 323.394,A -85,B 0,C 180,E1 -26248.382,E2 -26248.382} C_VEL
LIN {X 0,Y 136.25,Z 318.148,A -85,B 0,C 180,E1 -26252.339,E2 -26252.339} C_VEL
LIN {X 0,Y 134.464,Z 313.167,A -85,B 0,C 180,E1 -26256.92,E2 -26256.92} C_VEL
LIN {X 0,Y 133.373,Z 310.211,A -85,B 0,C 180,E1 -26259.969,E2 -26259.969} C_VEL
LIN {X 0,Y 132.419,Z 307.819,A -85,B 0,C 180,E1 -26262.793,E2 -26262.793} C_VEL
LIN {X 0,Y 130.939,Z 304.782,A -85,B 0,C 180,E1 -26267.602,E2 -26267.602} C_VEL
LIN {X 0,Y 130.118,Z 303.44,A -85,B 0,C 180,E1 -26270.674,E2 -26270.674} C_VEL
LIN {X 0,Y 129.347,Z 300.613,A -85,B 0,C 180,E1 -26280,E2 -26280} C_VEL
LIN {X 0,Y 129.216,Z 301.176,A -85,B 0,C 180,E1 -26283.117,E2 -26283.117} C_VEL
LIN {X 0,Y 129.237,Z 302.329,A -85,B 0,C 180,E1 -26286.244,E2 -26286.244} C_VEL
LIN {X 0,Y 130.672,Z 307.747,A -85,B 0,C 180,E1 -26295.6,E2 -26295.6} C_VEL
LIN {X 0,Y 132.471,Z 313.436,A -85,B 0,C 180,E1 -26301.8,E2 -26301.8} C_VEL
LIN {X 0,Y 134.027,Z 319.885,A -85,B 0,C 180,E1 -26306.956,E2 -26306.956} C_VEL
LIN {X 0,Y 135.423,Z 325.978,A -85,B 0,C 180,E1 -26311.263,E2 -26311.263} C_VEL
LIN {X 0,Y 136.499,Z 332.536,A -85,B 0,C 180,E1 -26315.397,E2 -26315.397} C_VEL
LIN {X 0,Y 136.819,Z 336.373,A -85,B 0,C 180,E1 -26317.588,E2 -26317.588} C_VEL
LIN {X 0,Y 134.924,Z 344.088,A -85,B 0,C 180,E1 -26320.957,E2 -26320.957} C_VEL
LIN {X 0,Y 132.11,Z 352.025,A -85,B 0,C 180,E1 -26324.63,E2 -26324.63} C_VEL
LIN {X 0,Y 129.769,Z 357.414,A -85,B 0,C 180,E1 -26327.399,E2 -26327.399} C_VEL
LIN {X 0,Y 125.935,Z 362.671,A -85,B 0,C 180,E1 -26330.082,E2 -26330.082} C_VEL
LIN {X 0,Y 120.472,Z 369.301,A -85,B 0,C 180,E1 -26334.318,E2 -26334.318} C_VEL
LIN {X 0,Y 115.81,Z 374.612,A -85,B 0,C 180,E1 -26338.953,E2 -26338.953} C_VEL
LIN {X 0,Y 111.863,Z 378.76,A -85,B 0,C 180,E1 -26343.916,E2 -26343.916} C_VEL
LIN {X 0,Y 109.689,Z 380.947,A -85,B 0,C 180,E1 -26347.398,E2 -26347.398} C_VEL
LIN {X 0,Y 106.739,Z 384.021,A -85,B 0,C 180,E1 -26354.736,E2 -26354.736} C_VEL
LIN {X 0,Y 105.901,Z 384.97,A -85,B 0,C 180,E1 -26358.522,E2 -26358.522} C_VEL
LIN {X 0,Y 105.504,Z 385.504,A -85,B 0,C 180,E1 -26362.35,E2 -26362.35} C_VEL
LIN {X 0,Y 105.49,Z 385.568,A -85,B 0,C 180,E1 -26367.91,E2 -26367.91} C_VEL
LIN {X 0,Y 105.676,Z 385.351,A -85,B 0,C 180,E1 -26370.006,E2 -26370.006} C_VEL
LIN {X 0,Y 105.501,Z 384.642,A -85,B 0,C 180,E1 -26373.825,E2 -26373.825} C_VEL
LIN {X 0,Y 105.527,Z 383.504,A -85,B 0,C 180,E1 -26377.66,E2 -26377.66} C_VEL
LIN {X 0,Y 106.297,Z 380.993,A -85,B 0,C 180,E1 -26383.386,E2 -26383.386} C_VEL
LIN {X 0,Y 107.917,Z 377.459,A -85,B 0,C 180,E1 -26389.009,E2 -26389.009} C_VEL
LIN {X 0,Y 110.622,Z 372.838,A -85,B 0,C 180,E1 -26394.396,E2 -26394.396} C_VEL
LIN {X 0,Y 114.142,Z 366.965,A -85,B 0,C 180,E1 -26399.516,E2 -26399.516} C_VEL
LIN {X 0,Y 116.846,Z 362.235,A -85,B 0,C 180,E1 -26402.78,E2 -26402.78} C_VEL
LIN {X 0,Y 120.9,Z 355.314,A -85,B 0,C 180,E1 -26406.578,E2 -26406.578} C_VEL
LIN {X 0,Y 123.041,Z 350.459,A -85,B 0,C 180,E1 -26408.931,E2 -26408.931} C_VEL
LIN {X 0,Y 125.679,Z 341.374,A -85,B 0,C 180,E1 -26412.944,E2 -26412.944} C_VEL
LIN {X 0,Y 127.634,Z 332.08,A -85,B 0,C 180,E1 -26416.492,E2 -26416.492} C_VEL
LIN {X 0,Y 128.744,Z 322.531,A -85,B 0,C 180,E1 -26419.846,E2 -26419.846} C_VEL
LIN {X 0,Y 128.496,Z 319.596,A -85,B 0,C 180,E1 -26421.023,E2 -26421.023} C_VEL
LIN {X 0,Y 126.737,Z 312.604,A -85,B 0,C 180,E1 -26424.391,E2 -26424.391} C_VEL
LIN {X 0,Y 124.164,Z 304.891,A -85,B 0,C 180,E1 -26428.5,E2 -26428.5} C_VEL
LIN {X 0,Y 122.054,Z 299.804,A -85,B 0,C 180,E1 -26431.638,E2 -26431.638} C_VEL
LIN {X 0,Y 119.99,Z 294.97,A -85,B 0,C 180,E1 -26434.872,E2 -26434.872} C_VEL
LIN {X 0,Y 117.72,Z 290.997,A -85,B 0,C 180,E1 -26438.322,E2 -26438.322} C_VEL
LIN {X 0,Y 117.042,Z 288.855,A -85,B 0,C 180,E1 -26439.802,E2 -26439.802} C_VEL
LIN {X 0,Y 114.474,Z 285.397,A -85,B 0,C 180,E1 -26444.305,E2 -26444.305} C_VEL
LIN {X 0,Y 113.288,Z 281.999,A -85,B 0,C 180,E1 -26447.648,E2 -26447.648} C_VEL
LIN {X 0,Y 110.959,Z 279.618,A -85,B 0,C 180,E1 -26454.549,E2 -26454.549} C_VEL
LIN {X 0,Y 110.207,Z 278.198,A -85,B 0,C 180,E1 -26460,E2 -26460} C_VEL
LIN {X 0,Y 111.097,Z 279.881,A -85,B 0,C 180,E1 -26471.911,E2 -26471.911} C_VEL
LIN {X 0,Y 112.596,Z 280.827,A -85,B 0,C 180,E1 -26476.41,E2 -26476.41} C_VEL
LIN {X 0,Y 113.342,Z 281.685,A -85,B 0,C 180,E1 -26478.294,E2 -26478.294} C_VEL
LIN {X 0,Y 114.184,Z 284.326,A -85,B 0,C 180,E1 -26480.903,E2 -26480.903} C_VEL
LIN {X 0,Y 114.711,Z 287.89,A -85,B 0,C 180,E1 -26483.274,E2 -26483.274} C_VEL
LIN {X 0,Y 115.674,Z 295.737,A -85,B 0,C 180,E1 -26488.001,E2 -26488.001} C_VEL
LIN {X 0,Y 116.354,Z 297.88,A -85,B 0,C 180,E1 -26489.694,E2 -26489.694} C_VEL
LIN {X 0,Y 118.793,Z 302.722,A -85,B 0,C 180,E1 -26494.071,E2 -26494.071} C_VEL
LIN {X 0,Y 121.775,Z 309.744,A -85,B 0,C 180,E1 -26499.409,E2 -26499.409} C_VEL
LIN {X 0,Y 123.581,Z 315.263,A -85,B 0,C 180,E1 -26503.035,E2 -26503.035} C_VEL
LIN {X 0,Y 124.749,Z 320.744,A -85,B 0,C 180,E1 -26506.257,E2 -26506.257} C_VEL
LIN {X 0,Y 124.644,Z 327.971,A -85,B 0,C 180,E1 -26509.902,E2 -26509.902} C_VEL
LIN {X 0,Y 124.061,Z 331.272,A -85,B 0,C 180,E1 -26511.448,E2 -26511.448} C_VEL
LIN {X 0,Y 119.225,Z 340.179,A -85,B 0,C 180,E1 -26514.913,E2 -26514.913} C_VEL
LIN {X 0,Y 113.942,Z 348.876,A -85,B 0,C 180,E1 -26519.406,E2 -26519.406} C_VEL
LIN {X 0,Y 109.862,Z 355.319,A -85,B 0,C 180,E1 -26523.923,E2 -26523.923} C_VEL
LIN {X 0,Y 106.217,Z 360.546,A -85,B 0,C 180,E1 -26528.653,E2 -26528.653} C_VEL
LIN {X 0,Y 102.945,Z 365.122,A -85,B 0,C 180,E1 -26534.147,E2 -26534.147} C_VEL
LIN {X 0,Y 101.324,Z 367.547,A -85,B 0,C 180,E1 -26537.984,E2 -26537.984} C_VEL
LIN {X 0,Y 100.101,Z 369.523,A -85,B 0,C 180,E1 -26541.922,E2 -26541.922} C_VEL
LIN {X 0,Y 99.298,Z 371.09,A -85,B 0,C 180,E1 -26545.935,E2 -26545.935} C_VEL
LIN {X 0,Y 98.85,Z 372.257,A -85,B 0,C 180,E1 -26549.994,E2 -26549.994} C_VEL
LIN {X 0,Y 98.769,Z 373.105,A -85,B 0,C 180,E1 -26554.996,E2 -26554.996} C_VEL
LIN {X 0,Y 99.501,Z 373.347,A -85,B 0,C 180,E1 -26562.227,E2 -26562.227} C_VEL
LIN {X 0,Y 100.412,Z 372.953,A -85,B 0,C 180,E1 -26566.252,E2 -26566.252} C_VEL
LIN {X 0,Y 103.45,Z 370.906,A -85,B 0,C 180,E1 -26574.049,E2 -26574.049} C_VEL
LIN {X 0,Y 106.92,Z 368.284,A -85,B 0,C 180,E1 -26579.53,E2 -26579.53} C_VEL
LIN {X 0,Y 111.208,Z 364.585,A -85,B 0,C 180,E1 -26584.758,E2 -26584.758} C_VEL
LIN {X 0,Y 116.125,Z 359.888,A -85,B 0,C 180,E1 -26589.448,E2 -26589.448} C_VEL
LIN {X 0,Y 121.836,Z 353.853,A -85,B 0,C 180,E1 -26593.798,E2 -26593.798} C_VEL
LIN {X 0,Y 128.111,Z 346.326,A -85,B 0,C 180,E1 -26597.775,E2 -26597.775} C_VEL
LIN {X 0,Y 131.055,Z 342.334,A -85,B 0,C 180,E1 -26599.474,E2 -26599.474} C_VEL
LIN {X 0,Y 131.754,Z 340.865,A -85,B 0,C 180,E1 -26600.2,E2 -26600.2} C_VEL
LIN {X 0,Y 132.552,Z 336.138,A -85,B 0,C 180,E1 -26603.234,E2 -26603.234} C_VEL
LIN {X 0,Y 132.541,Z 330.709,A -85,B 0,C 180,E1 -26607.077,E2 -26607.077} C_VEL
LIN {X 0,Y 131.872,Z 325.208,A -85,B 0,C 180,E1 -26611.337,E2 -26611.337} C_VEL
LIN {X 0,Y 131.093,Z 321.492,A -85,B 0,C 180,E1 -26614.603,E2 -26614.603} C_VEL
LIN {X 0,Y 129.747,Z 316.883,A -85,B 0,C 180,E1 -26619.385,E2 -26619.385} C_VEL
LIN {X 0,Y 128.977,Z 314.499,A -85,B 0,C 180,E1 -26622.319,E2 -26622.319} C_VEL
LIN {X 0,Y 127.682,Z 311.41,A -85,B 0,C 180,E1 -26627.28,E2 -26627.28} C_VEL
LIN {X 0,Y 127.035,Z 309.967,A -85,B 0,C 180,E1 -26630.446,E2 -26630.446} C_VEL
LIN {X 0,Y 126.493,Z 307.161,A -85,B 0,C 180,E1 -26640.118,E2 -26640.118} C_VEL
LIN {X 0,Y 126.325,Z 307.786,A -85,B 0,C 180,E1 -26643.189,E2 -26643.189} C_VEL
LIN {X 0,Y 126.233,Z 309.039,A -85,B 0,C 180,E1 -26646.393,E2 -26646.393} C_VEL
LIN {X 0,Y 127.082,Z 313.522,A -85,B 0,C 180,E1 -26654.41,E2 -26654.41} C_VEL
LIN {X 0,Y 128.451,Z 318.926,A -85,B 0,C 180,E1 -26660.834,E2 -26660.834} C_VEL
LIN {X 0,Y 129.725,Z 326.003,A -85,B 0,C 180,E1 -26666.883,E2 -26666.883} C_VEL
LIN {X 0,Y 130.642,Z 332.246,A -85,B 0,C 180,E1 -26671.497,E2 -26671.497} C_VEL
LIN {X 0,Y 131.192,Z 338.002,A -85,B 0,C 180,E1 -26675.364,E2 -26675.364} C_VEL
LIN {X 0,Y 131.106,Z 339.953,A -85,B 0,C 180,E1 -26676.487,E2 -26676.487} C_VEL
LIN {X 0,Y 128.637,Z 347.611,A -85,B 0,C 180,E1 -26680.111,E2 -26680.111} C_VEL
LIN {X 0,Y 125.118,Z 355.713,A -85,B 0,C 180,E1 -26684.267,E2 -26684.267} C_VEL
LIN {X 0,Y 123.605,Z 358.549,A -85,B 0,C 180,E1 -26685.859,E2 -26685.859} C_VEL
LIN {X 0,Y 117.542,Z 365.898,A -85,B 0,C 180,E1 -26690.009,E2 -26690.009} C_VEL
LIN {X 0,Y 111.311,Z 372.661,A -85,B 0,C 180,E1 -26695.379,E2 -26695.379} C_VEL
LIN {X 0,Y 106.787,Z 377.154,A -85,B 0,C 180,E1 -26700.429,E2 -26700.429} C_VEL
LIN {X 0,Y 103.156,Z 380.583,A -85,B 0,C 180,E1 -26705.878,E2 -26705.878} C_VEL
LIN {X 0,Y 101.217,Z 382.302,A -85,B 0,C 180,E1 -26709.692,E2 -26709.692} C_VEL
LIN {X 0,Y 98.927,Z 384.57,A -85,B 0,C 180,E1 -26717.701,E2 -26717.701} C_VEL
LIN {X 0,Y 98.448,Z 385.081,A -85,B 0,C 180,E1 -26721.798,E2 -26721.798} C_VEL
LIN {X 0,Y 98.442,Z 385.104,A -85,B 0,C 180,E1 -26728.165,E2 -26728.165} C_VEL
LIN {X 0,Y 98.455,Z 384.594,A -85,B 0,C 180,E1 -26732.049,E2 -26732.049} C_VEL
LIN {X 0,Y 98.485,Z 383.022,A -85,B 0,C 180,E1 -26738.211,E2 -26738.211} C_VEL
LIN {X 0,Y 99.367,Z 380.49,A -85,B 0,C 180,E1 -26744.338,E2 -26744.338} C_VEL
LIN {X 0,Y 101.188,Z 376.932,A -85,B 0,C 180,E1 -26750.327,E2 -26750.327} C_VEL
LIN {X 0,Y 104.147,Z 372.279,A -85,B 0,C 180,E1 -26756.023,E2 -26756.023} C_VEL
LIN {X 0,Y 107.907,Z 366.363,A -85,B 0,C 180,E1 -26761.408,E2 -26761.408} C_VEL
LIN {X 0,Y 111.764,Z 360.36,A -85,B 0,C 180,E1 -26765.574,E2 -26765.574} C_VEL
LIN {X 0,Y 116.018,Z 353.124,A -85,B 0,C 180,E1 -26769.505,E2 -26769.505} C_VEL
LIN {X 0,Y 119.14,Z 344.131,A -85,B 0,C 180,E1 -26773.885,E2 -26773.885} C_VEL
LIN {X 0,Y 121.46,Z 335.368,A -85,B 0,C 180,E1 -26777.561,E2 -26777.561} C_VEL
LIN {X 0,Y 123.092,Z 326.091,A -85,B 0,C 180,E1 -26781.094,E2 -26781.094} C_VEL
LIN {X 0,Y 123.109,Z 323.316,A -85,B 0,C 180,E1 -26782.261,E2 -26782.261} C_VEL
LIN {X 0,Y 121.705,Z 316.611,A -85,B 0,C 180,E1 -26785.811,E2 -26785.811} C_VEL
LIN {X 0,Y 119.601,Z 309.388,A -85,B 0,C 180,E1 -26790.035,E2 -26790.035} C_VEL
LIN {X 0,Y 117.593,Z 304.031,A -85,B 0,C 180,E1 -26793.71,E2 -26793.71} C_VEL
LIN {X 0,Y 116.501,Z 300.801,A -85,B 0,C 180,E1 -26795.971,E2 -26795.971} C_VEL
LIN {X 0,Y 114.324,Z 295.963,A -85,B 0,C 180,E1 -26800.239,E2 -26800.239} C_VEL
LIN {X 0,Y 112.672,Z 293.084,A -85,B 0,C 180,E1 -26803.699,E2 -26803.699} C_VEL
LIN {X 0,Y 111.119,Z 288.725,A -85,B 0,C 180,E1 -26808.485,E2 -26808.485} C_VEL
LIN {X 0,Y 109.361,Z 286.581,A -85,B 0,C 180,E1 -26814.469,E2 -26814.469} C_VEL
LIN {X 0,Y 108.637,Z 285.188,A -85,B 0,C 180,E1 -26820,E2 -26820} C_VEL
LIN {X 0,Y 109.147,Z 286.627,A -85,B 0,C 180,E1 -26831.138,E2 -26831.138} C_VEL
LIN {X 0,Y 110.71,Z 287.861,A -85,B 0,C 180,E1 -26836.481,E2 -26836.481} C_VEL
LIN {X 0,Y 111.736,Z 290.777,A -85,B 0,C 180,E1 -26840.238,E2 -26840.238} C_VEL
LIN {X 0,Y 113.432,Z 292.542,A -85,B 0,C 180,E1 -26843.749,E2 -26843.749} C_VEL
LIN {X 0,Y 116.354,Z 297.88,A -85,B 0,C 180,E1 -26849.694,E2 -26849.694} C_VEL
LIN {X 0,Y 117.294,Z 301.14,A -85,B 0,C 180,E1 -26852.07,E2 -26852.07} C_VEL
LIN {X 0,Y 117.687,Z 305.089,A -85,B 0,C 180,E1 -26854.235,E2 -26854.235} C_VEL
LIN {X 0,Y 117.781,Z 316.273,A -85,B 0,C 180,E1 -26859.863,E2 -26859.863} C_VEL
LIN {X 0,Y 118.15,Z 318.697,A -85,B 0,C 180,E1 -26861.413,E2 -26861.413} C_VEL
LIN {X 0,Y 118.928,Z 322.108,A -85,B 0,C 180,E1 -26863.724,E2 -26863.724} C_VEL
LIN {X 0,Y 119.124,Z 325.741,A -85,B 0,C 180,E1 -26865.868,E2 -26865.868} C_VEL
LIN {X 0,Y 118.51,Z 332.02,A -85,B 0,C 180,E1 -26869.276,E2 -26869.276} C_VEL
LIN {X 0,Y 115.54,Z 337.532,A -85,B 0,C 180,E1 -26871.423,E2 -26871.423} C_VEL
LIN {X 0,Y 110.648,Z 345.423,A -85,B 0,C 180,E1 -26875.129,E2 -26875.129} C_VEL
LIN {X 0,Y 105.559,Z 353.051,A -85,B 0,C 180,E1 -26879.944,E2 -26879.944} C_VEL
LIN {X 0,Y 100.948,Z 359.327,A -85,B 0,C 180,E1 -26885.303,E2 -26885.303} C_VEL
LIN {X 0,Y 97.248,Z 364.246,A -85,B 0,C 180,E1 -26891.015,E2 -26891.015} C_VEL
LIN {X 0,Y 94.434,Z 368.056,A -85,B 0,C 180,E1 -26897.093,E2 -26897.093} C_VEL
LIN {X 0,Y 93.12,Z 370.018,A -85,B 0,C 180,E1 -26901.312,E2 -26901.312} C_VEL
LIN {X 0,Y 92.238,Z 371.574,A -85,B 0,C 180,E1 -26905.624,E2 -26905.624} C_VEL
LIN {X 0,Y 91.772,Z 372.717,A -85,B 0,C 180,E1 -26909.994,E2 -26909.994} C_VEL
LIN {X 0,Y 91.698,Z 373.494,A -85,B 0,C 180,E1 -26914.884,E2 -26914.884} C_VEL
LIN {X 0,Y 92.568,Z 373.768,A -85,B 0,C 180,E1 -26923.159,E2 -26923.159} C_VEL
LIN {X 0,Y 93.586,Z 373.355,A -85,B 0,C 180,E1 -26927.474,E2 -26927.474} C_VEL
LIN {X 0,Y 96.976,Z 371.277,A -85,B 0,C 180,E1 -26935.768,E2 -26935.768} C_VEL
LIN {X 0,Y 100.771,Z 368.629,A -85,B 0,C 180,E1 -26941.531,E2 -26941.531} C_VEL
LIN {X 0,Y 105.342,Z 364.966,A -85,B 0,C 180,E1 -26946.894,E2 -26946.894} C_VEL
LIN {X 0,Y 110.714,Z 360.174,A -85,B 0,C 180,E1 -26951.792,E2 -26951.792} C_VEL
LIN {X 0,Y 116.796,Z 354.106,A -85,B 0,C 180,E1 -26956.219,E2 -26956.219} C_VEL
LIN {X 0,Y 123.433,Z 346.535,A -85,B 0,C 180,E1 -26960.226,E2 -26960.226} C_VEL
LIN {X 0,Y 125.696,Z 343.586,A -85,B 0,C 180,E1 -26961.507,E2 -26961.507} C_VEL
LIN {X 0,Y 126.53,Z 340.824,A -85,B 0,C 180,E1 -26963.338,E2 -26963.338} C_VEL
LIN {X 0,Y 127.022,Z 336.712,A -85,B 0,C 180,E1 -26966.406,E2 -26966.406} C_VEL
LIN {X 0,Y 126.923,Z 331.117,A -85,B 0,C 180,E1 -26971.02,E2 -26971.02} C_VEL
LIN {X 0,Y 126.353,Z 326.595,A -85,B 0,C 180,E1 -26975.243,E2 -26975.243} C_VEL
LIN {X 0,Y 125.355,Z 322.086,A -85,B 0,C 180,E1 -26980.342,E2 -26980.342} C_VEL
LIN {X 0,Y 124.733,Z 319.697,A -85,B 0,C 180,E1 -26983.636,E2 -26983.636} C_VEL
LIN {X 0,Y 124.07,Z 317.809,A -85,B 0,C 180,E1 -26986.904,E2 -26986.904} C_VEL
LIN {X 0,Y 123.56,Z 316.329,A -85,B 0,C 180,E1 -26990.175,E2 -26990.175} C_VEL
LIN {X 0,Y 123.25,Z 313.513,A -85,B 0,C 180,E1 -27000,E2 -27000} C_VEL
LIN {X 0,Y 123.031,Z 314.211,A -85,B 0,C 180,E1 -27003.274,E2 -27003.274} C_VEL
LIN {X 0,Y 122.84,Z 315.587,A -85,B 0,C 180,E1 -27006.57,E2 -27006.57} C_VEL
LIN {X 0,Y 123.441,Z 319.968,A -85,B 0,C 180,E1 -27014.582,E2 -27014.582} C_VEL
LIN {X 0,Y 124.209,Z 324.232,A -85,B 0,C 180,E1 -27019.846,E2 -27019.846} C_VEL
LIN {X 0,Y 124.929,Z 330.701,A -85,B 0,C 180,E1 -27025.841,E2 -27025.841} C_VEL
LIN {X 0,Y 125.419,Z 336.202,A -85,B 0,C 180,E1 -27030.286,E2 -27030.286} C_VEL
LIN {X 0,Y 125.606,Z 341.278,A -85,B 0,C 180,E1 -27034.023,E2 -27034.023} C_VEL
LIN {X 0,Y 125.142,Z 343.761,A -85,B 0,C 180,E1 -27035.476,E2 -27035.476} C_VEL
LIN {X 0,Y 122.153,Z 351.094,A -85,B 0,C 180,E1 -27039.262,E2 -27039.262} C_VEL
LIN {X 0,Y 118.424,Z 358.312,A -85,B 0,C 180,E1 -27043.373,E2 -27043.373} C_VEL
LIN {X 0,Y 115.376,Z 362.175,A -85,B 0,C 180,E1 -27045.54,E2 -27045.54} C_VEL
LIN {X 0,Y 109.198,Z 368.738,A -85,B 0,C 180,E1 -27049.947,E2 -27049.947} C_VEL
LIN {X 0,Y 103.812,Z 373.984,A -85,B 0,C 180,E1 -27054.876,E2 -27054.876} C_VEL
LIN {X 0,Y 99.209,Z 378.079,A -85,B 0,C 180,E1 -27060.279,E2 -27060.279} C_VEL
LIN {X 0,Y 96.678,Z 380.218,A -85,B 0,C 180,E1 -27064.147,E2 -27064.147} C_VEL
LIN {X 0,Y 93.019,Z 383.242,A -85,B 0,C 180,E1 -27072.416,E2 -27072.416} C_VEL
LIN {X 0,Y 91.986,Z 384.167,A -85,B 0,C 180,E1 -27076.756,E2 -27076.756} C_VEL
LIN {X 0,Y 91.393,Z 384.657,A -85,B 0,C 180,E1 -27081.16,E2 -27081.16} C_VEL
LIN {X 0,Y 91.392,Z 384.606,A -85,B 0,C 180,E1 -27088.568,E2 -27088.568} C_VEL
LIN {X 0,Y 91.404,Z 384.23,A -85,B 0,C 180,E1 -27091.712,E2 -27091.712} C_VEL
LIN {X 0,Y 91.425,Z 382.539,A -85,B 0,C 180,E1 -27098.85,E2 -27098.85} C_VEL
LIN {X 0,Y 92.452,Z 379.982,A -85,B 0,C 180,E1 -27105.437,E2 -27105.437} C_VEL
LIN {X 0,Y 94.52,Z 376.4,A -85,B 0,C 180,E1 -27111.832,E2 -27111.832} C_VEL
LIN {X 0,Y 97.772,Z 371.717,A -85,B 0,C 180,E1 -27117.861,E2 -27117.861} C_VEL
LIN {X 0,Y 101.81,Z 365.762,A -85,B 0,C 180,E1 -27123.528,E2 -27123.528} C_VEL
LIN {X 0,Y 106.968,Z 358.365,A -85,B 0,C 180,E1 -27128.628,E2 -27128.628} C_VEL
LIN {X 0,Y 110.41,Z 352.432,A -85,B 0,C 180,E1 -27131.948,E2 -27131.948} C_VEL
LIN {X 0,Y 113.575,Z 344.017,A -85,B 0,C 180,E1 -27136.24,E2 -27136.24} C_VEL
LIN {X 0,Y 116.011,Z 335.778,A -85,B 0,C 180,E1 -27139.897,E2 -27139.897} C_VEL
LIN {X 0,Y 117.669,Z 327.435,A -85,B 0,C 180,E1 -27143.326,E2 -27143.326} C_VEL
LIN {X 0,Y 116.664,Z 320.728,A -85,B 0,C 180,E1 -27147.169,E2 -27147.169} C_VEL
LIN {X 0,Y 114.874,Z 313.442,A -85,B 0,C 180,E1 -27151.874,E2 -27151.874} C_VEL
LIN {X 0,Y 112.786,Z 306.507,A -85,B 0,C 180,E1 -27157.08,E2 -27157.08} C_VEL
LIN {X 0,Y 110.799,Z 301.226,A -85,B 0,C 180,E1 -27162.09,E2 -27162.09} C_VEL
LIN {X 0,Y 108.679,Z 295.847,A -85,B 0,C 180,E1 -27168.814,E2 -27168.814} C_VEL
LIN {X 0,Y 107.75,Z 294.005,A -85,B 0,C 180,E1 -27172.505,E2 -27172.505} C_VEL
LIN {X 0,Y 106.657,Z 292.092,A -85,B 0,C 180,E1 -27180,E2 -27180} C_VEL
LIN {X 0,Y 106.629,Z 292.96,A -85,B 0,C 180,E1 -27188.602,E2 -27188.602} C_VEL
LIN {X 0,Y 108.023,Z 294.191,A -85,B 0,C 180,E1 -27195.085,E2 -27195.085} C_VEL
LIN {X 0,Y 108.776,Z 296.697,A -85,B 0,C 180,E1 -27198.848,E2 -27198.848} C_VEL
LIN {X 0,Y 110.155,Z 298.612,A -85,B 0,C 180,E1 -27202.508,E2 -27202.508} C_VEL
LIN {X 0,Y 112.639,Z 303.585,A -85,B 0,C 180,E1 -27208.667,E2 -27208.667} C_VEL
LIN {X 0,Y 114.365,Z 307.467,A -85,B 0,C 180,E1 -27212.529,E2 -27212.529} C_VEL
LIN {X 0,Y 116.44,Z 312.902,A -85,B 0,C 180,E1 -27217.127,E2 -27217.127} C_VEL
LIN {X 0,Y 118.15,Z 318.697,A -85,B 0,C 180,E1 -27221.413,E2 -27221.413} C_VEL
LIN {X 0,Y 118.317,Z 321.236,A -85,B 0,C 180,E1 -27222.89,E2 -27222.89} C_VEL
LIN {X 0,Y 117.28,Z 325.673,A -85,B 0,C 180,E1 -27224.784,E2 -27224.784} C_VEL
LIN {X 0,Y 115.238,Z 330.285,A -85,B 0,C 180,E1 -27226.429,E2 -27226.429} C_VEL
LIN {X 0,Y 111.513,Z 336.4,A -85,B 0,C 180,E1 -27228.541,E2 -27228.541} C_VEL
LIN {X 0,Y 107.595,Z 342.147,A -85,B 0,C 180,E1 -27230.898,E2 -27230.898} C_VEL
LIN {X 0,Y 102.051,Z 350.138,A -85,B 0,C 180,E1 -27235.372,E2 -27235.372} C_VEL
LIN {X 0,Y 97.756,Z 355.953,A -85,B 0,C 180,E1 -27239.778,E2 -27239.778} C_VEL
LIN {X 0,Y 93.214,Z 361.673,A -85,B 0,C 180,E1 -27245.494,E2 -27245.494} C_VEL
LIN {X 0,Y 89.46,Z 366.186,A -85,B 0,C 180,E1 -27251.678,E2 -27251.678} C_VEL
LIN {X 0,Y 87.571,Z 368.564,A -85,B 0,C 180,E1 -27256.061,E2 -27256.061} C_VEL
LIN {X 0,Y 86.129,Z 370.514,A -85,B 0,C 180,E1 -27260.601,E2 -27260.601} C_VEL
LIN {X 0,Y 85.182,Z 372.057,A -85,B 0,C 180,E1 -27265.26,E2 -27265.26} C_VEL
LIN {X 0,Y 84.676,Z 373.176,A -85,B 0,C 180,E1 -27269.993,E2 -27269.993} C_VEL
LIN {X 0,Y 84.629,Z 373.884,A -85,B 0,C 180,E1 -27274.757,E2 -27274.757} C_VEL
LIN {X 0,Y 85.651,Z 374.191,A -85,B 0,C 180,E1 -27284.243,E2 -27284.243} C_VEL
LIN {X 0,Y 86.821,Z 373.754,A -85,B 0,C 180,E1 -27288.885,E2 -27288.885} C_VEL
LIN {X 0,Y 90.601,Z 371.65,A -85,B 0,C 180,E1 -27297.73,E2 -27297.73} C_VEL
LIN {X 0,Y 94.761,Z 368.975,A -85,B 0,C 180,E1 -27303.789,E2 -27303.789} C_VEL
LIN {X 0,Y 99.718,Z 365.284,A -85,B 0,C 180,E1 -27309.361,E2 -27309.361} C_VEL
LIN {X 0,Y 105.493,Z 360.462,A -85,B 0,C 180,E1 -27314.38,E2 -27314.38} C_VEL
LIN {X 0,Y 111.973,Z 354.36,A -85,B 0,C 180,E1 -27318.858,E2 -27318.858} C_VEL
LIN {X 0,Y 118.876,Z 346.877,A -85,B 0,C 180,E1 -27322.807,E2 -27322.807} C_VEL
LIN {X 0,Y 120.029,Z 345.454,A -85,B 0,C 180,E1 -27323.426,E2 -27323.426} C_VEL
LIN {X 0,Y 121.048,Z 342.272,A -85,B 0,C 180,E1 -27325.815,E2 -27325.815} C_VEL
LIN {X 0,Y 121.575,Z 337.319,A -85,B 0,C 180,E1 -27330.115,E2 -27330.115} C_VEL
LIN {X 0,Y 121.552,Z 332.995,A -85,B 0,C 180,E1 -27334.301,E2 -27334.301} C_VEL
LIN {X 0,Y 120.967,Z 328.495,A -85,B 0,C 180,E1 -27339.598,E2 -27339.598} C_VEL
LIN {X 0,Y 120.588,Z 325.922,A -85,B 0,C 180,E1 -27343.057,E2 -27343.057} C_VEL
LIN {X 0,Y 120.103,Z 324.024,A -85,B 0,C 180,E1 -27346.463,E2 -27346.463} C_VEL
LIN {X 0,Y 119.711,Z 322.475,A -85,B 0,C 180,E1 -27349.855,E2 -27349.855} C_VEL
LIN {X 0,Y 119.655,Z 319.693,A -85,B 0,C 180,E1 -27360,E2 -27360} C_VEL
LIN {X 0,Y 119.362,Z 320.493,A -85,B 0,C 180,E1 -27363.375,E2 -27363.375} C_VEL
LIN {X 0,Y 119.035,Z 323.669,A -85,B 0,C 180,E1 -27370.202,E2 -27370.202} C_VEL
LIN {X 0,Y 119.339,Z 325.431,A -85,B 0,C 180,E1 -27373.625,E2 -27373.625} C_VEL
LIN {X 0,Y 119.725,Z 329.361,A -85,B 0,C 180,E1 -27378.837,E2 -27378.837} C_VEL
LIN {X 0,Y 119.961,Z 334.639,A -85,B 0,C 180,E1 -27384.211,E2 -27384.211} C_VEL
LIN {X 0,Y 120.088,Z 339.58,A -85,B 0,C 180,E1 -27388.626,E2 -27388.626} C_VEL
LIN {X 0,Y 120.044,Z 343.441,A -85,B 0,C 180,E1 -27391.796,E2 -27391.796} C_VEL
LIN {X 0,Y 119.863,Z 345.285,A -85,B 0,C 180,E1 -27393.214,E2 -27393.214} C_VEL
LIN {X 0,Y 117.729,Z 350.247,A -85,B 0,C 180,E1 -27395.988,E2 -27395.988} C_VEL
LIN {X 0,Y 113.385,Z 358.07,A -85,B 0,C 180,E1 -27400.606,E2 -27400.606} C_VEL
LIN {X 0,Y 111.525,Z 360.686,A -85,B 0,C 180,E1 -27402.238,E2 -27402.238} C_VEL
LIN {X 0,Y 104.874,Z 367.439,A -85,B 0,C 180,E1 -27406.624,E2 -27406.624} C_VEL
LIN {X 0,Y 98.933,Z 372.874,A -85,B 0,C 180,E1 -27411.602,E2 -27411.602} C_VEL
LIN {X 0,Y 93.07,Z 377.737,A -85,B 0,C 180,E1 -27418.097,E2 -27418.097} C_VEL
LIN {X 0,Y 90.308,Z 379.854,A -85,B 0,C 180,E1 -27422.172,E2 -27422.172} C_VEL
LIN {X 0,Y 87.964,Z 381.549,A -85,B 0,C 180,E1 -27426.462,E2 -27426.462} C_VEL
LIN {X 0,Y 85.049,Z 383.76,A -85,B 0,C 180,E1 -27435.654,E2 -27435.654} C_VEL
LIN {X 0,Y 84.187,Z 384.321,A -85,B 0,C 180,E1 -27445.218,E2 -27445.218} C_VEL
LIN {X 0,Y 84.351,Z 383.9,A -85,B 0,C 180,E1 -27451.08,E2 -27451.08} C_VEL
LIN {X 0,Y 84.395,Z 382.057,A -85,B 0,C 180,E1 -27459.594,E2 -27459.594} C_VEL
LIN {X 0,Y 85.582,Z 379.473,A -85,B 0,C 180,E1 -27466.711,E2 -27466.711} C_VEL
LIN {X 0,Y 87.928,Z 375.866,A -85,B 0,C 180,E1 -27473.563,E2 -27473.563} C_VEL
LIN {X 0,Y 91.518,Z 371.153,A -85,B 0,C 180,E1 -27479.952,E2 -27479.952} C_VEL
LIN {X 0,Y 95.141,Z 366.279,A -85,B 0,C 180,E1 -27484.931,E2 -27484.931} C_VEL
LIN {X 0,Y 99.54,Z 360.403,A -85,B 0,C 180,E1 -27489.46,E2 -27489.46} C_VEL
LIN {X 0,Y 103.386,Z 354.862,A -85,B 0,C 180,E1 -27492.834,E2 -27492.834} C_VEL
LIN {X 0,Y 106.402,Z 348.317,A -85,B 0,C 180,E1 -27496.607,E2 -27496.607} C_VEL
LIN {X 0,Y 109.727,Z 339.475,A -85,B 0,C 180,E1 -27500.958,E2 -27500.958} C_VEL
LIN {X 0,Y 112.012,Z 331.178,A -85,B 0,C 180,E1 -27504.661,E2 -27504.661} C_VEL
LIN {X 0,Y 111.998,Z 328.508,A -85,B 0,C 180,E1 -27506.163,E2 -27506.163} C_VEL
LIN {X 0,Y 111.036,Z 321.598,A -85,B 0,C 180,E1 -27510.729,E2 -27510.729} C_VEL
LIN {X 0,Y 109.703,Z 315.421,A -85,B 0,C 180,E1 -27515.392,E2 -27515.392} C_VEL
LIN {X 0,Y 108.536,Z 311.129,A -85,B 0,C 180,E1 -27519.137,E2 -27519.137} C_VEL
LIN {X 0,Y 107.361,Z 307.023,A -85,B 0,C 180,E1 -27523.277,E2 -27523.277} C_VEL
LIN {X 0,Y 105.674,Z 301.791,A -85,B 0,C 180,E1 -27530.43,E2 -27530.43} C_VEL
LIN {X 0,Y 105.279,Z 300.897,A -85,B 0,C 180,E1 -27532.328,E2 -27532.328} C_VEL
LIN {X 0,Y 104.279,Z 298.83,A -85,B 0,C 180,E1 -27540,E2 -27540} C_VEL
LIN {X 0,Y 104.1,Z 299.513,A -85,B 0,C 180,E1 -27547.761,E2 -27547.761} C_VEL
LIN {X 0,Y 104.619,Z 300.131,A -85,B 0,C 180,E1 -27551.627,E2 -27551.627} C_VEL
LIN {X 0,Y 105.351,Z 301.325,A -85,B 0,C 180,E1 -27555.477,E2 -27555.477} C_VEL
LIN {X 0,Y 107.263,Z 305.719,A -85,B 0,C 180,E1 -27563.15,E2 -27563.15} C_VEL
LIN {X 0,Y 108.895,Z 309.59,A -85,B 0,C 180,E1 -27568.105,E2 -27568.105} C_VEL
LIN {X 0,Y 110.513,Z 314.008,A -85,B 0,C 180,E1 -27572.722,E2 -27572.722} C_VEL
LIN {X 0,Y 112.171,Z 319.532,A -85,B 0,C 180,E1 -27577.653,E2 -27577.653} C_VEL
LIN {X 0,Y 113.268,Z 324.988,A -85,B 0,C 180,E1 -27581.87,E2 -27581.87} C_VEL
LIN {X 0,Y 113.477,Z 328.204,A -85,B 0,C 180,E1 -27584.058,E2 -27584.058} C_VEL
LIN {X 0,Y 112.958,Z 332.791,A -85,B 0,C 180,E1 -27586.805,E2 -27586.805} C_VEL
LIN {X 0,Y 112.317,Z 334.66,A -85,B 0,C 180,E1 -27587.721,E2 -27587.721} C_VEL
LIN {X 0,Y 107.595,Z 342.147,A -85,B 0,C 180,E1 -27590.898,E2 -27590.898} C_VEL
LIN {X 0,Y 104.488,Z 346.026,A -85,B 0,C 180,E1 -27592.631,E2 -27592.631} C_VEL
LIN {X 0,Y 98.048,Z 351.938,A -85,B 0,C 180,E1 -27595.283,E2 -27595.283} C_VEL
LIN {X 0,Y 91.584,Z 357.297,A -85,B 0,C 180,E1 -27598.514,E2 -27598.514} C_VEL
LIN {X 0,Y 88.558,Z 360.17,A -85,B 0,C 180,E1 -27601.162,E2 -27601.162} C_VEL
LIN {X 0,Y 83.998,Z 365.32,A -85,B 0,C 180,E1 -27607.875,E2 -27607.875} C_VEL
LIN {X 0,Y 80.721,Z 369.073,A -85,B 0,C 180,E1 -27614.851,E2 -27614.851} C_VEL
LIN {X 0,Y 79.156,Z 371.01,A -85,B 0,C 180,E1 -27619.764,E2 -27619.764} C_VEL
LIN {X 0,Y 78.132,Z 372.539,A -85,B 0,C 180,E1 -27624.832,E2 -27624.832} C_VEL
LIN {X 0,Y 77.535,Z 374.253,A -85,B 0,C 180,E1 -27634.373,E2 -27634.373} C_VEL
LIN {X 0,Y 77.916,Z 374.659,A -85,B 0,C 180,E1 -27640.385,E2 -27640.385} C_VEL
LIN {X 0,Y 78.764,Z 374.614,A -85,B 0,C 180,E1 -27645.519,E2 -27645.519} C_VEL
LIN {X 0,Y 80.095,Z 374.152,A -85,B 0,C 180,E1 -27650.539,E2 -27650.539} C_VEL
LIN {X 0,Y 84.35,Z 372.023,A -85,B 0,C 180,E1 -27659.986,E2 -27659.986} C_VEL
LIN {X 0,Y 88.919,Z 369.321,A -85,B 0,C 180,E1 -27666.347,E2 -27666.347} C_VEL
LIN {X 0,Y 94.313,Z 365.602,A -85,B 0,C 180,E1 -27672.109,E2 -27672.109} C_VEL
LIN {X 0,Y 100.52,Z 360.749,A -85,B 0,C 180,E1 -27677.224,E2 -27677.224} C_VEL
LIN {X 0,Y 107.407,Z 354.614,A -85,B 0,C 180,E1 -27681.73,E2 -27681.73} C_VEL
LIN {X 0,Y 114.601,Z 347.192,A -85,B 0,C 180,E1 -27685.601,E2 -27685.601} C_VEL
LIN {X 0,Y 115.59,Z 344.063,A -85,B 0,C 180,E1 -27688.334,E2 -27688.334} C_VEL
LIN {X 0,Y 116.183,Z 339.384,A -85,B 0,C 180,E1 -27693.019,E2 -27693.019} C_VEL
LIN {X 0,Y 116.296,Z 336.175,A -85,B 0,C 180,E1 -27696.647,E2 -27696.647} C_VEL
LIN {X 0,Y 116.035,Z 332.002,A -85,B 0,C 180,E1 -27702.371,E2 -27702.371} C_VEL
LIN {X 0,Y 115.747,Z 329.853,A -85,B 0,C 180,E1 -27706.265,E2 -27706.265} C_VEL
LIN {X 0,Y 115.509,Z 328.441,A -85,B 0,C 180,E1 -27709.482,E2 -27709.482} C_VEL
LIN {X 0,Y 115.378,Z 326.438,A -85,B 0,C 180,E1 -27716.507,E2 -27716.507} C_VEL
LIN {X 0,Y 115.736,Z 325.659,A -85,B 0,C 180,E1 -27720,E2 -27720} C_VEL
LIN {X 0,Y 115.35,Z 326.572,A -85,B 0,C 180,E1 -27723.493,E2 -27723.493} C_VEL
LIN {X 0,Y 114.909,Z 330.38,A -85,B 0,C 180,E1 -27731.905,E2 -27731.905} C_VEL
LIN {X 0,Y 115.024,Z 334.286,A -85,B 0,C 180,E1 -27737.788,E2 -27737.788} C_VEL
LIN {X 0,Y 114.88,Z 339.353,A -85,B 0,C 180,E1 -27743.429,E2 -27743.429} C_VEL
LIN {X 0,Y 114.551,Z 344.867,A -85,B 0,C 180,E1 -27748.724,E2 -27748.724} C_VEL
LIN {X 0,Y 114.373,Z 347.045,A -85,B 0,C 180,E1 -27750.664,E2 -27750.664} C_VEL
LIN {X 0,Y 113.91,Z 348.752,A -85,B 0,C 180,E1 -27751.98,E2 -27751.98} C_VEL
LIN {X 0,Y 110.424,Z 355.043,A -85,B 0,C 180,E1 -27755.769,E2 -27755.769} C_VEL
LIN {X 0,Y 106.786,Z 360.435,A -85,B 0,C 180,E1 -27759.357,E2 -27759.357} C_VEL
LIN {X 0,Y 99.806,Z 367.159,A -85,B 0,C 180,E1 -27763.808,E2 -27763.808} C_VEL
LIN {X 0,Y 92.871,Z 373.03,A -85,B 0,C 180,E1 -27769.394,E2 -27769.394} C_VEL
LIN {X 0,Y 87.091,Z 377.392,A -85,B 0,C 180,E1 -27775.614,E2 -27775.614} C_VEL
LIN {X 0,Y 84.067,Z 379.49,A -85,B 0,C 180,E1 -27779.902,E2 -27779.902} C_VEL
LIN {X 0,Y 81.467,Z 381.173,A -85,B 0,C 180,E1 -27784.456,E2 -27784.456} C_VEL
LIN {X 0,Y 79.538,Z 382.466,A -85,B 0,C 180,E1 -27789.31,E2 -27789.31} C_VEL
LIN {X 0,Y 78.161,Z 383.351,A -85,B 0,C 180,E1 -27794.359,E2 -27794.359} C_VEL
LIN {X 0,Y 77.092,Z 383.886,A -85,B 0,C 180,E1 -27804.777,E2 -27804.777} C_VEL
LIN {X 0,Y 77.312,Z 383.519,A -85,B 0,C 180,E1 -27810.592,E2 -27810.592} C_VEL
LIN {X 0,Y 77.118,Z 382.8,A -85,B 0,C 180,E1 -27815.236,E2 -27815.236} C_VEL
LIN {X 0,Y 77.373,Z 381.573,A -85,B 0,C 180,E1 -27820.474,E2 -27820.474} C_VEL
LIN {X 0,Y 78.774,Z 378.964,A -85,B 0,C 180,E1 -27828.203,E2 -27828.203} C_VEL
LIN {X 0,Y 81.431,Z 375.33,A -85,B 0,C 180,E1 -27835.573,E2 -27835.573} C_VEL
LIN {X 0,Y 85.394,Z 370.588,A -85,B 0,C 180,E1 -27842.349,E2 -27842.349} C_VEL
LIN {X 0,Y 89.305,Z 365.687,A -85,B 0,C 180,E1 -27847.59,E2 -27847.59} C_VEL
LIN {X 0,Y 95.179,Z 358.473,A -85,B 0,C 180,E1 -27853.088,E2 -27853.088} C_VEL
LIN {X 0,Y 98.132,Z 354.193,A -85,B 0,C 180,E1 -27855.748,E2 -27855.748} C_VEL
LIN {X 0,Y 102.455,Z 345.114,A -85,B 0,C 180,E1 -27861.028,E2 -27861.028} C_VEL
LIN {X 0,Y 105.773,Z 336.189,A -85,B 0,C 180,E1 -27865.47,E2 -27865.47} C_VEL
LIN {X 0,Y 106.592,Z 332.891,A -85,B 0,C 180,E1 -27867.125,E2 -27867.125} C_VEL
LIN {X 0,Y 106.197,Z 326.988,A -85,B 0,C 180,E1 -27871.327,E2 -27871.327} C_VEL
LIN {X 0,Y 105.505,Z 321.859,A -85,B 0,C 180,E1 -27875.397,E2 -27875.397} C_VEL
LIN {X 0,Y 104.488,Z 316.491,A -85,B 0,C 180,E1 -27880.348,E2 -27880.348} C_VEL
LIN {X 0,Y 103.727,Z 312.866,A -85,B 0,C 180,E1 -27884.276,E2 -27884.276} C_VEL
LIN {X 0,Y 102.442,Z 307.622,A -85,B 0,C 180,E1 -27892.114,E2 -27892.114} C_VEL
LIN {X 0,Y 101.544,Z 305.413,A -85,B 0,C 180,E1 -27900,E2 -27900} C_VEL
LIN {X 0,Y 101.318,Z 306.079,A -85,B 0,C 180,E1 -27907.975,E2 -27907.975} C_VEL
LIN {X 0,Y 101.751,Z 306.766,A -85,B 0,C 180,E1 -27911.96,E2 -27911.96} C_VEL
LIN {X 0,Y 102.248,Z 308.283,A -85,B 0,C 180,E1 -27915.959,E2 -27915.959} C_VEL
LIN {X 0,Y 103.483,Z 311.347,A -85,B 0,C 180,E1 -27921.934,E2 -27921.934} C_VEL
LIN {X 0,Y 104.474,Z 314.095,A -85,B 0,C 180,E1 -27925.93,E2 -27925.93} C_VEL
LIN {X 0,Y 105.518,Z 317.464,A -85,B 0,C 180,E1 -27930.008,E2 -27930.008} C_VEL
LIN {X 0,Y 107.05,Z 323.682,A -85,B 0,C 180,E1 -27936.219,E2 -27936.219} C_VEL
LIN {X 0,Y 107.801,Z 328.896,A -85,B 0,C 180,E1 -27940.689,E2 -27940.689} C_VEL
LIN {X 0,Y 107.789,Z 331.746,A -85,B 0,C 180,E1 -27942.781,E2 -27942.781} C_VEL
LIN {X 0,Y 107.091,Z 335.4,A -85,B 0,C 180,E1 -27945.124,E2 -27945.124} C_VEL
LIN {X 0,Y 101.531,Z 343.792,A -85,B 0,C 180,E1 -27948.876,E2 -27948.876} C_VEL
LIN {X 0,Y 95.331,Z 351.979,A -85,B 0,C 180,E1 -27953.852,E2 -27953.852} C_VEL
LIN {X 0,Y 89.989,Z 358.565,A -85,B 0,C 180,E1 -27959.486,E2 -27959.486} C_VEL
LIN {X 0,Y 88.558,Z 360.17,A -85,B 0,C 180,E1 -27961.162,E2 -27961.162} C_VEL
LIN {X 0,Y 85.635,Z 362.874,A -85,B 0,C 180,E1 -27964.051,E2 -27964.051} C_VEL
LIN {X 0,Y 77.246,Z 368.108,A -85,B 0,C 180,E1 -27970.965,E2 -27970.965} C_VEL
LIN {X 0,Y 73.344,Z 370.522,A -85,B 0,C 180,E1 -27975.898,E2 -27975.898} C_VEL
LIN {X 0,Y 72.209,Z 371.5,A -85,B 0,C 180,E1 -27978.75,E2 -27978.75} C_VEL
LIN {X 0,Y 71.089,Z 373.019,A -85,B 0,C 180,E1 -27984.318,E2 -27984.318} C_VEL
LIN {X 0,Y 70.465,Z 374.641,A -85,B 0,C 180,E1 -27994.14,E2 -27994.14} C_VEL
LIN {X 0,Y 70.929,Z 375.094,A -85,B 0,C 180,E1 -28001.421,E2 -28001.421} C_VEL
LIN {X 0,Y 71.936,Z 375.034,A -85,B 0,C 180,E1 -28007.035,E2 -28007.035} C_VEL
LIN {X 0,Y 75.6,Z 373.667,A -85,B 0,C 180,E1 -28017.689,E2 -28017.689} C_VEL
LIN {X 0,Y 78.256,Z 372.395,A -85,B 0,C 180,E1 -28022.596,E2 -28022.596} C_VEL
LIN {X 0,Y 83.268,Z 369.668,A -85,B 0,C 180,E1 -28029.264,E2 -28029.264} C_VEL
LIN {X 0,Y 89.151,Z 365.919,A -85,B 0,C 180,E1 -28035.184,E2 -28035.184} C_VEL
LIN {X 0,Y 95.825,Z 361.036,A -85,B 0,C 180,E1 -28040.352,E2 -28040.352} C_VEL
LIN {X 0,Y 103.131,Z 354.869,A -85,B 0,C 180,E1 -28044.85,E2 -28044.85} C_VEL
LIN {X 0,Y 109.18,Z 348.973,A -85,B 0,C 180,E1 -28047.958,E2 -28047.958} C_VEL
LIN {X 0,Y 110.21,Z 345.635,A -85,B 0,C 180,E1 -28051.429,E2 -28051.429} C_VEL
LIN {X 0,Y 110.933,Z 341.457,A -85,B 0,C 180,E1 -28056.368,E2 -28056.368} C_VEL
LIN {X 0,Y 111.081,Z 337.852,A -85,B 0,C 180,E1 -28061.61,E2 -28061.61} C_VEL
LIN {X 0,Y 111.021,Z 335.785,A -85,B 0,C 180,E1 -28065.332,E2 -28065.332} C_VEL
LIN {X 0,Y 110.972,Z 334.181,A -85,B 0,C 180,E1 -28069.047,E2 -28069.047} C_VEL
LIN {X 0,Y 111.012,Z 332.144,A -85,B 0,C 180,E1 -28076.37,E2 -28076.37} C_VEL
LIN {X 0,Y 111.462,Z 331.422,A -85,B 0,C 180,E1 -28080,E2 -28080} C_VEL
LIN {X 0,Y 110.957,Z 332.407,A -85,B 0,C 180,E1 -28083.631,E2 -28083.631} C_VEL
LIN {X 0,Y 110.345,Z 335.558,A -85,B 0,C 180,E1 -28091.015,E2 -28091.015} C_VEL
LIN {X 0,Y 110.128,Z 339.093,A -85,B 0,C 180,E1 -28096.833,E2 -28096.833} C_VEL
LIN {X 0,Y 109.589,Z 343.866,A -85,B 0,C 180,E1 -28102.63,E2 -28102.63} C_VEL
LIN {X 0,Y 108.877,Z 348.833,A -85,B 0,C 180,E1 -28107.846,E2 -28107.846} C_VEL
LIN {X 0,Y 108.162,Z 351.535,A -85,B 0,C 180,E1 -28110.287,E2 -28110.287} C_VEL
LIN {X 0,Y 104.05,Z 357.678,A -85,B 0,C 180,E1 -28114.293,E2 -28114.293} C_VEL
LIN {X 0,Y 101.172,Z 361.432,A -85,B 0,C 180,E1 -28116.989,E2 -28116.989} C_VEL
LIN {X 0,Y 93.818,Z 367.878,A -85,B 0,C 180,E1 -28121.497,E2 -28121.497} C_VEL
LIN {X 0,Y 86.967,Z 373.139,A -85,B 0,C 180,E1 -28126.88,E2 -28126.88} C_VEL
LIN {X 0,Y 81.305,Z 377.044,A -85,B 0,C 180,E1 -28132.775,E2 -28132.775} C_VEL
LIN {X 0,Y 77.982,Z 379.127,A -85,B 0,C 180,E1 -28137.275,E2 -28137.275} C_VEL
LIN {X 0,Y 75.091,Z 380.797,A -85,B 0,C 180,E1 -28142.107,E2 -28142.107} C_VEL
LIN {X 0,Y 72.901,Z 382.078,A -85,B 0,C 180,E1 -28147.327,E2 -28147.327} C_VEL
LIN {X 0,Y 71.332,Z 382.94,A -85,B 0,C 180,E1 -28152.817,E2 -28152.817} C_VEL
LIN {X 0,Y 70.029,Z 383.452,A -85,B 0,C 180,E1 -28164.249,E2 -28164.249} C_VEL
LIN {X 0,Y 70.279,Z 383.131,A -85,B 0,C 180,E1 -28170.008,E2 -28170.008} C_VEL
LIN {X 0,Y 70.047,Z 382.334,A -85,B 0,C 180,E1 -28175.767,E2 -28175.767} C_VEL
LIN {X 0,Y 70.371,Z 381.09,A -85,B 0,C 180,E1 -28181.53,E2 -28181.53} C_VEL
LIN {X 0,Y 72.039,Z 378.455,A -85,B 0,C 180,E1 -28189.974,E2 -28189.974} C_VEL
LIN {X 0,Y 75.057,Z 374.794,A -85,B 0,C 180,E1 -28197.925,E2 -28197.925} C_VEL
LIN {X 0,Y 79.435,Z 370.021,A -85,B 0,C 180,E1 -28205.114,E2 -28205.114} C_VEL
LIN {X 0,Y 85.112,Z 363.506,A -85,B 0,C 180,E1 -28211.999,E2 -28211.999} C_VEL
LIN {X 0,Y 91.155,Z 356.463,A -85,B 0,C 180,E1 -28217.101,E2 -28217.101} C_VEL
LIN {X 0,Y 93.948,Z 351.966,A -85,B 0,C 180,E1 -28220.075,E2 -28220.075} C_VEL
LIN {X 0,Y 98.252,Z 343.368,A -85,B 0,C 180,E1 -28225.094,E2 -28225.094} C_VEL
LIN {X 0,Y 101.083,Z 336.105,A -85,B 0,C 180,E1 -28228.884,E2 -28228.884} C_VEL
LIN {X 0,Y 101.075,Z 330.698,A -85,B 0,C 180,E1 -28233.133,E2 -28233.133} C_VEL
LIN {X 0,Y 100.601,Z 324.764,A -85,B 0,C 180,E1 -28238.484,E2 -28238.484} C_VEL
LIN {X 0,Y 100.126,Z 321.163,A -85,B 0,C 180,E1 -28242.25,E2 -28242.25} C_VEL
LIN {X 0,Y 99.769,Z 318.225,A -85,B 0,C 180,E1 -28245.727,E2 -28245.727} C_VEL
LIN {X 0,Y 99.14,Z 314.272,A -85,B 0,C 180,E1 -28251.85,E2 -28251.85} C_VEL
LIN {X 0,Y 98.692,Z 312.812,A -85,B 0,C 180,E1 -28255.917,E2 -28255.917} C_VEL
LIN {X 0,Y 98.404,Z 311.84,A -85,B 0,C 180,E1 -28260.431,E2 -28260.431} C_VEL
LIN {X 0,Y 98.142,Z 312.472,A -85,B 0,C 180,E1 -28268.235,E2 -28268.235} C_VEL
LIN {X 0,Y 98.472,Z 313.259,A -85,B 0,C 180,E1 -28272.364,E2 -28272.364} C_VEL
LIN {X 0,Y 98.857,Z 314.893,A -85,B 0,C 180,E1 -28276.522,E2 -28276.522} C_VEL
LIN {X 0,Y 99.5,Z 316.853,A -85,B 0,C 180,E1 -28280.682,E2 -28280.682} C_VEL
